LIN {X 0,Y 524.415,Z 426.256,A -85,B 0,C 180,E1 -4599.936,E2 -4599.936} C_VEL
LIN {X 0,Y 524.541,Z 418.004,A -85,B 0,C 180,E1 -4600.323,E2 -4600.323} C_VEL
LIN {X 0,Y 524.652,Z 409.12,A -85,B 0,C 180,E1 -4600.638,E2 -4600.638} C_VEL
LIN {X 0,Y 524.801,Z 400.246,A -85,B 0,C 180,E1 -4600.855,E2 -4600.855} C_VEL
LIN {X 0,Y 524.849,Z 331.396,A -85,B 0,C 180,E1 -4601.818,E2 -4601.818} C_VEL
LIN {X 0,Y 523.839,Z 323.933,A -85,B 0,C 180,E1 -4601.968,E2 -4601.968} C_VEL
LIN {X 0,Y 523.832,Z 321.449,A -85,B 0,C 180,E1 -4602.396,E2 -4602.396} C_VEL
LIN {X 0,Y 524.033,Z 307.521,A -85,B 0,C 180,E1 -4605.213,E2 -4605.213} C_VEL
LIN {X 0,Y 524.371,Z 292.162,A -85,B 0,C 180,E1 -4608.358,E2 -4608.358} C_VEL
LIN {X 0,Y 524.384,Z 283.062,A -85,B 0,C 180,E1 -4610.254,E2 -4610.254} C_VEL
LIN {X 0,Y 523.979,Z 280.14,A -85,B 0,C 180,E1 -4610.923,E2 -4610.923} C_VEL
LIN {X 0,Y 523.931,Z 280.033,A -85,B 0,C 180,E1 -4614.196,E2 -4614.196} C_VEL
LIN {X 0,Y 523.899,Z 280.036,A -85,B 0,C 180,E1 -4617.135,E2 -4617.135} C_VEL
LIN {X 0,Y 523.893,Z 280.04,A -85,B 0,C 180,E1 -4619.758,E2 -4619.758} C_VEL
LIN {X 0,Y 523.929,Z 280.029,A -85,B 0,C 180,E1 -4622.449,E2 -4622.449} C_VEL
LIN {X 0,Y 523.909,Z 280.038,A -85,B 0,C 180,E1 -4625.227,E2 -4625.227} C_VEL
LIN {X 0,Y 523.907,Z 280.033,A -85,B 0,C 180,E1 -4628.102,E2 -4628.102} C_VEL
LIN {X 0,Y 523.914,Z 280.04,A -85,B 0,C 180,E1 -4631.305,E2 -4631.305} C_VEL
LIN {X 0,Y 523.927,Z 280.032,A -85,B 0,C 180,E1 -4634.688,E2 -4634.688} C_VEL
LIN {X 0,Y 523.892,Z 280.035,A -85,B 0,C 180,E1 -4637.875,E2 -4637.875} C_VEL
LIN {X 0,Y 523.904,Z 280.041,A -85,B 0,C 180,E1 -4641.081,E2 -4641.081} C_VEL
LIN {X 0,Y 523.885,Z 280.035,A -85,B 0,C 180,E1 -4643.824,E2 -4643.824} C_VEL
LIN {X 0,Y 523.903,Z 280.038,A -85,B 0,C 180,E1 -4646.633,E2 -4646.633} C_VEL
LIN {X 0,Y 523.928,Z 280.031,A -85,B 0,C 180,E1 -4649.354,E2 -4649.354} C_VEL
LIN {X 0,Y 523.908,Z 280.035,A -85,B 0,C 180,E1 -4652.293,E2 -4652.293} C_VEL
LIN {X 0,Y 523.892,Z 280.035,A -85,B 0,C 180,E1 -4655.426,E2 -4655.426} C_VEL
LIN {X 0,Y 523.922,Z 280.032,A -85,B 0,C 180,E1 -4657.939,E2 -4657.939} C_VEL
LIN {X 0,Y 523.94,Z 280.036,A -85,B 0,C 180,E1 -4660.406,E2 -4660.406} C_VEL
LIN {X 0,Y 523.883,Z 280.039,A -85,B 0,C 180,E1 -4662.834,E2 -4662.834} C_VEL
LIN {X 0,Y 523.951,Z 280.027,A -85,B 0,C 180,E1 -4665.235,E2 -4665.235} C_VEL
LIN {X 0,Y 524.002,Z 280.028,A -85,B 0,C 180,E1 -4668.394,E2 -4668.394} C_VEL
LIN {X 0,Y 523.971,Z 280.025,A -85,B 0,C 180,E1 -4671.515,E2 -4671.515} C_VEL
LIN {X 0,Y 524.022,Z 280.021,A -85,B 0,C 180,E1 -4674.613,E2 -4674.613} C_VEL
LIN {X 0,Y 524.093,Z 280.013,A -85,B 0,C 180,E1 -4677.694,E2 -4677.694} C_VEL
LIN {X 0,Y 524.085,Z 280.019,A -85,B 0,C 180,E1 -4680,E2 -4680} C_VEL
LIN {X 0,Y 524.092,Z 280.013,A -85,B 0,C 180,E1 -4682.306,E2 -4682.306} C_VEL
LIN {X 0,Y 523.997,Z 280.026,A -85,B 0,C 180,E1 -4686.16,E2 -4686.16} C_VEL
LIN {X 0,Y 523.932,Z 280.031,A -85,B 0,C 180,E1 -4689.263,E2 -4689.263} C_VEL
LIN {X 0,Y 523.933,Z 280.03,A -85,B 0,C 180,E1 -4692.393,E2 -4692.393} C_VEL
LIN {X 0,Y 523.9,Z 280.041,A -85,B 0,C 180,E1 -4695.563,E2 -4695.563} C_VEL
LIN {X 0,Y 523.901,Z 280.036,A -85,B 0,C 180,E1 -4697.971,E2 -4697.971} C_VEL
LIN {X 0,Y 523.931,Z 280.029,A -85,B 0,C 180,E1 -4700.412,E2 -4700.412} C_VEL
LIN {X 0,Y 523.875,Z 280.038,A -85,B 0,C 180,E1 -4702.895,E2 -4702.895} C_VEL
LIN {X 0,Y 523.887,Z 280.043,A -85,B 0,C 180,E1 -4705.422,E2 -4705.422} C_VEL
LIN {X 0,Y 523.886,Z 280.036,A -85,B 0,C 180,E1 -4708.004,E2 -4708.004} C_VEL
LIN {X 0,Y 523.897,Z 280.037,A -85,B 0,C 180,E1 -4710.848,E2 -4710.848} C_VEL
LIN {X 0,Y 523.916,Z 280.033,A -85,B 0,C 180,E1 -4713.729,E2 -4713.729} C_VEL
LIN {X 0,Y 523.878,Z 280.037,A -85,B 0,C 180,E1 -4716.399,E2 -4716.399} C_VEL
LIN {X 0,Y 523.902,Z 280.042,A -85,B 0,C 180,E1 -4719.086,E2 -4719.086} C_VEL
LIN {X 0,Y 523.887,Z 280.035,A -85,B 0,C 180,E1 -4722.125,E2 -4722.125} C_VEL
LIN {X 0,Y 523.926,Z 280.033,A -85,B 0,C 180,E1 -4725.312,E2 -4725.312} C_VEL
LIN {X 0,Y 523.908,Z 280.04,A -85,B 0,C 180,E1 -4728.696,E2 -4728.696} C_VEL
LIN {X 0,Y 523.904,Z 280.033,A -85,B 0,C 180,E1 -4731.898,E2 -4731.898} C_VEL
LIN {X 0,Y 523.91,Z 280.037,A -85,B 0,C 180,E1 -4734.913,E2 -4734.913} C_VEL
LIN {X 0,Y 523.926,Z 280.03,A -85,B 0,C 180,E1 -4737.681,E2 -4737.681} C_VEL
LIN {X 0,Y 523.931,Z 280.036,A -85,B 0,C 180,E1 -4740.681,E2 -4740.681} C_VEL
LIN {X 0,Y 523.896,Z 280.034,A -85,B 0,C 180,E1 -4743.725,E2 -4743.725} C_VEL
LIN {X 0,Y 523.902,Z 280.034,A -85,B 0,C 180,E1 -4746.27,E2 -4746.27} C_VEL
LIN {X 0,Y 523.993,Z 280.189,A -85,B 0,C 180,E1 -4749.155,E2 -4749.155} C_VEL
LIN {X 0,Y 524.495,Z 286.09,A -85,B 0,C 180,E1 -4750.429,E2 -4750.429} C_VEL
LIN {X 0,Y 524.172,Z 299.754,A -85,B 0,C 180,E1 -4753.246,E2 -4753.246} C_VEL
LIN {X 0,Y 523.917,Z 313.418,A -85,B 0,C 180,E1 -4756.028,E2 -4756.028} C_VEL
LIN {X 0,Y 523.85,Z 323.715,A -85,B 0,C 180,E1 -4758.064,E2 -4758.064} C_VEL
LIN {X 0,Y 524.395,Z 328.212,A -85,B 0,C 180,E1 -4758.173,E2 -4758.173} C_VEL
LIN {X 0,Y 524.964,Z 334.33,A -85,B 0,C 180,E1 -4758.27,E2 -4758.27} C_VEL
LIN {X 0,Y 524.799,Z 399.153,A -85,B 0,C 180,E1 -4759.17,E2 -4759.17} C_VEL
LIN {X 0,Y 524.672,Z 408.418,A -85,B 0,C 180,E1 -4759.387,E2 -4759.387} C_VEL
LIN {X 0,Y 524.591,Z 416.888,A -85,B 0,C 180,E1 -4759.678,E2 -4759.678} C_VEL
LIN {X 0,Y 524.418,Z 425.391,A -85,B 0,C 180,E1 -4760.064,E2 -4760.064} C_VEL
LIN {X 0,Y 524.239,Z 433.724,A -85,B 0,C 180,E1 -4760.548,E2 -4760.548} C_VEL
LIN {X 0,Y 524.099,Z 441.761,A -85,B 0,C 180,E1 -4761.129,E2 -4761.129} C_VEL
LIN {X 0,Y 523.896,Z 450.433,A -85,B 0,C 180,E1 -4761.903,E2 -4761.903} C_VEL
LIN {X 0,Y 523.729,Z 458.939,A -85,B 0,C 180,E1 -4762.87,E2 -4762.87} C_VEL
LIN {X 0,Y 523.639,Z 465.61,A -85,B 0,C 180,E1 -4763.836,E2 -4763.836} C_VEL
LIN {X 0,Y 523.484,Z 469.989,A -85,B 0,C 180,E1 -4764.608,E2 -4764.608} C_VEL
LIN {X 0,Y 523.469,Z 475.15,A -85,B 0,C 180,E1 -4765.765,E2 -4765.765} C_VEL
LIN {X 0,Y 523.379,Z 478.938,A -85,B 0,C 180,E1 -4766.921,E2 -4766.921} C_VEL
LIN {X 0,Y 523.336,Z 480.68,A -85,B 0,C 180,E1 -4767.691,E2 -4767.691} C_VEL
LIN {X 0,Y 523.273,Z 481.928,A -85,B 0,C 180,E1 -4768.461,E2 -4768.461} C_VEL
LIN {X 0,Y 523.246,Z 482.706,A -85,B 0,C 180,E1 -4769.23,E2 -4769.23} C_VEL
LIN {X 0,Y 523.243,Z 483,A -85,B 0,C 180,E1 -4770,E2 -4770} C_VEL
LIN {X 0,Y 523.246,Z 482.705,A -85,B 0,C 180,E1 -4770.77,E2 -4770.77} C_VEL
LIN {X 0,Y 523.273,Z 481.927,A -85,B 0,C 180,E1 -4771.539,E2 -4771.539} C_VEL
LIN {X 0,Y 523.336,Z 480.679,A -85,B 0,C 180,E1 -4772.309,E2 -4772.309} C_VEL
LIN {X 0,Y 523.407,Z 477.786,A -85,B 0,C 180,E1 -4773.464,E2 -4773.464} C_VEL
LIN {X 0,Y 523.469,Z 475.149,A -85,B 0,C 180,E1 -4774.235,E2 -4774.235} C_VEL
LIN {X 0,Y 523.484,Z 469.986,A -85,B 0,C 180,E1 -4775.392,E2 -4775.392} C_VEL
LIN {X 0,Y 523.667,Z 463.738,A -85,B 0,C 180,E1 -4776.468,E2 -4776.468} C_VEL
LIN {X 0,Y 523.757,Z 455.74,A -85,B 0,C 180,E1 -4777.517,E2 -4777.517} C_VEL
LIN {X 0,Y 523.931,Z 448.398,A -85,B 0,C 180,E1 -4778.291,E2 -4778.291} C_VEL
LIN {X 0,Y 524.12,Z 440.535,A -85,B 0,C 180,E1 -4778.968,E2 -4778.968} C_VEL
LIN {X 0,Y 524.265,Z 432.224,A -85,B 0,C 180,E1 -4779.549,E2 -4779.549} C_VEL
LIN {X 0,Y 524.478,Z 421.614,A -85,B 0,C 180,E1 -4780.129,E2 -4780.129} C_VEL
LIN {X 0,Y 524.626,Z 410.084,A -85,B 0,C 180,E1 -4780.565,E2 -4780.565} C_VEL
LIN {X 0,Y 524.715,Z 400.451,A -85,B 0,C 180,E1 -4780.808,E2 -4780.808} C_VEL
LIN {X 0,Y 524.955,Z 348.572,A -85,B 0,C 180,E1 -4781.536,E2 -4781.536} C_VEL
LIN {X 0,Y 524.78,Z 330.794,A -85,B 0,C 180,E1 -4781.783,E2 -4781.783} C_VEL
LIN {X 0,Y 523.845,Z 323.822,A -85,B 0,C 180,E1 -4781.929,E2 -4781.929} C_VEL
LIN {X 0,Y 523.879,Z 317.322,A -85,B 0,C 180,E1 -4783.183,E2 -4783.183} C_VEL
LIN {X 0,Y 524.104,Z 303.658,A -85,B 0,C 180,E1 -4785.955,E2 -4785.955} C_VEL
LIN {X 0,Y 524.412,Z 289.994,A -85,B 0,C 180,E1 -4788.762,E2 -4788.762} C_VEL
LIN {X 0,Y 524.299,Z 282.187,A -85,B 0,C 180,E1 -4790.396,E2 -4790.396} C_VEL
LIN {X 0,Y 523.975,Z 280.145,A -85,B 0,C 180,E1 -4790.871,E2 -4790.871} C_VEL
LIN {X 0,Y 523.93,Z 280.033,A -85,B 0,C 180,E1 -4794.196,E2 -4794.196} C_VEL
LIN {X 0,Y 523.897,Z 280.037,A -85,B 0,C 180,E1 -4797.135,E2 -4797.135} C_VEL
LIN {X 0,Y 523.889,Z 280.039,A -85,B 0,C 180,E1 -4799.758,E2 -4799.758} C_VEL
LIN {X 0,Y 523.925,Z 280.03,A -85,B 0,C 180,E1 -4802.449,E2 -4802.449} C_VEL
LIN {X 0,Y 523.904,Z 280.04,A -85,B 0,C 180,E1 -4805.227,E2 -4805.227} C_VEL
LIN {X 0,Y 523.904,Z 280.033,A -85,B 0,C 180,E1 -4808.102,E2 -4808.102} C_VEL
LIN {X 0,Y 523.913,Z 280.039,A -85,B 0,C 180,E1 -4811.305,E2 -4811.305} C_VEL
LIN {X 0,Y 523.926,Z 280.033,A -85,B 0,C 180,E1 -4814.688,E2 -4814.688} C_VEL
LIN {X 0,Y 523.89,Z 280.035,A -85,B 0,C 180,E1 -4817.875,E2 -4817.875} C_VEL
LIN {X 0,Y 523.903,Z 280.04,A -85,B 0,C 180,E1 -4821.081,E2 -4821.081} C_VEL
LIN {X 0,Y 523.869,Z 280.037,A -85,B 0,C 180,E1 -4823.823,E2 -4823.823} C_VEL
LIN {X 0,Y 523.902,Z 280.039,A -85,B 0,C 180,E1 -4826.633,E2 -4826.633} C_VEL
LIN {X 0,Y 523.927,Z 280.031,A -85,B 0,C 180,E1 -4829.354,E2 -4829.354} C_VEL
LIN {X 0,Y 523.907,Z 280.036,A -85,B 0,C 180,E1 -4832.294,E2 -4832.294} C_VEL
LIN {X 0,Y 523.891,Z 280.035,A -85,B 0,C 180,E1 -4835.426,E2 -4835.426} C_VEL
LIN {X 0,Y 523.921,Z 280.032,A -85,B 0,C 180,E1 -4837.939,E2 -4837.939} C_VEL
LIN {X 0,Y 523.94,Z 280.036,A -85,B 0,C 180,E1 -4840.407,E2 -4840.407} C_VEL
LIN {X 0,Y 523.882,Z 280.039,A -85,B 0,C 180,E1 -4842.834,E2 -4842.834} C_VEL
LIN {X 0,Y 523.951,Z 280.027,A -85,B 0,C 180,E1 -4845.235,E2 -4845.235} C_VEL
LIN {X 0,Y 524.002,Z 280.028,A -85,B 0,C 180,E1 -4848.394,E2 -4848.394} C_VEL
LIN {X 0,Y 523.941,Z 280.029,A -85,B 0,C 180,E1 -4851.515,E2 -4851.515} C_VEL
LIN {X 0,Y 524.022,Z 280.021,A -85,B 0,C 180,E1 -4854.613,E2 -4854.613} C_VEL
LIN {X 0,Y 524.093,Z 280.013,A -85,B 0,C 180,E1 -4857.694,E2 -4857.694} C_VEL
LIN {X 0,Y 524.085,Z 280.019,A -85,B 0,C 180,E1 -4860,E2 -4860} C_VEL
LIN {X 0,Y 524.092,Z 280.013,A -85,B 0,C 180,E1 -4862.306,E2 -4862.306} C_VEL
LIN {X 0,Y 523.997,Z 280.026,A -85,B 0,C 180,E1 -4866.16,E2 -4866.16} C_VEL
LIN {X 0,Y 523.932,Z 280.031,A -85,B 0,C 180,E1 -4869.263,E2 -4869.263} C_VEL
LIN {X 0,Y 523.933,Z 280.03,A -85,B 0,C 180,E1 -4872.393,E2 -4872.393} C_VEL
LIN {X 0,Y 523.9,Z 280.041,A -85,B 0,C 180,E1 -4875.563,E2 -4875.563} C_VEL
LIN {X 0,Y 523.913,Z 280.032,A -85,B 0,C 180,E1 -4878.781,E2 -4878.781} C_VEL
LIN {X 0,Y 523.911,Z 280.037,A -85,B 0,C 180,E1 -4881.235,E2 -4881.235} C_VEL
LIN {X 0,Y 523.891,Z 280.034,A -85,B 0,C 180,E1 -4884.574,E2 -4884.574} C_VEL
LIN {X 0,Y 523.901,Z 280.037,A -85,B 0,C 180,E1 -4887.705,E2 -4887.705} C_VEL
LIN {X 0,Y 523.899,Z 280.035,A -85,B 0,C 180,E1 -4890.648,E2 -4890.648} C_VEL
LIN {X 0,Y 523.903,Z 280.039,A -85,B 0,C 180,E1 -4893.367,E2 -4893.367} C_VEL
LIN {X 0,Y 523.878,Z 280.036,A -85,B 0,C 180,E1 -4896.399,E2 -4896.399} C_VEL
LIN {X 0,Y 523.902,Z 280.042,A -85,B 0,C 180,E1 -4899.087,E2 -4899.087} C_VEL
LIN {X 0,Y 523.888,Z 280.035,A -85,B 0,C 180,E1 -4902.125,E2 -4902.125} C_VEL
LIN {X 0,Y 523.927,Z 280.033,A -85,B 0,C 180,E1 -4905.312,E2 -4905.312} C_VEL
LIN {X 0,Y 523.872,Z 280.044,A -85,B 0,C 180,E1 -4906.871,E2 -4906.871} C_VEL
LIN {X 0,Y 523.184,Z 280.125,A -85,B 0,C 180,E1 -4907.512,E2 -4907.512} C_VEL
LIN {X 0,Y 520.321,Z 280.484,A -85,B 0,C 180,E1 -4908.554,E2 -4908.554} C_VEL
LIN {X 0,Y 517.928,Z 280.779,A -85,B 0,C 180,E1 -4909.392,E2 -4909.392} C_VEL
LIN {X 0,Y 516.922,Z 280.903,A -85,B 0,C 180,E1 -4910.04,E2 -4910.04} C_VEL
LIN {X 0,Y 516.851,Z 280.913,A -85,B 0,C 180,E1 -4910.259,E2 -4910.259} C_VEL
LIN {X 0,Y 516.845,Z 280.914,A -85,B 0,C 180,E1 -4913.252,E2 -4913.252} C_VEL
LIN {X 0,Y 516.875,Z 280.91,A -85,B 0,C 180,E1 -4916.119,E2 -4916.119} C_VEL
LIN {X 0,Y 516.875,Z 280.912,A -85,B 0,C 180,E1 -4918.939,E2 -4918.939} C_VEL
LIN {X 0,Y 516.858,Z 280.914,A -85,B 0,C 180,E1 -4922.109,E2 -4922.109} C_VEL
LIN {X 0,Y 516.843,Z 280.915,A -85,B 0,C 180,E1 -4925.069,E2 -4925.069} C_VEL
LIN {X 0,Y 516.869,Z 280.898,A -85,B 0,C 180,E1 -4927.622,E2 -4927.622} C_VEL
LIN {X 0,Y 516.925,Z 281.074,A -85,B 0,C 180,E1 -4929.091,E2 -4929.091} C_VEL
LIN {X 0,Y 517.472,Z 285.88,A -85,B 0,C 180,E1 -4930.152,E2 -4930.152} C_VEL
LIN {X 0,Y 517.255,Z 297.588,A -85,B 0,C 180,E1 -4932.608,E2 -4932.608} C_VEL
LIN {X 0,Y 516.908,Z 313.2,A -85,B 0,C 180,E1 -4935.834,E2 -4935.834} C_VEL
LIN {X 0,Y 516.779,Z 323.603,A -85,B 0,C 180,E1 -4937.928,E2 -4937.928} C_VEL
LIN {X 0,Y 516.978,Z 325.468,A -85,B 0,C 180,E1 -4938.008,E2 -4938.008} C_VEL
LIN {X 0,Y 518.064,Z 333.866,A -85,B 0,C 180,E1 -4938.15,E2 -4938.15} C_VEL
LIN {X 0,Y 517.841,Z 399.389,A -85,B 0,C 180,E1 -4939.072,E2 -4939.072} C_VEL
LIN {X 0,Y 517.699,Z 408.571,A -85,B 0,C 180,E1 -4939.292,E2 -4939.292} C_VEL
LIN {X 0,Y 517.566,Z 418.209,A -85,B 0,C 180,E1 -4939.635,E2 -4939.635} C_VEL
LIN {X 0,Y 517.426,Z 428.284,A -85,B 0,C 180,E1 -4940.126,E2 -4940.126} C_VEL
LIN {X 0,Y 517.146,Z 438.743,A -85,B 0,C 180,E1 -4940.812,E2 -4940.812} C_VEL
LIN {X 0,Y 516.908,Z 446.911,A -85,B 0,C 180,E1 -4941.497,E2 -4941.497} C_VEL
LIN {X 0,Y 516.744,Z 453.65,A -85,B 0,C 180,E1 -4942.183,E2 -4942.183} C_VEL
LIN {X 0,Y 516.66,Z 460.03,A -85,B 0,C 180,E1 -4942.968,E2 -4942.968} C_VEL
LIN {X 0,Y 516.585,Z 465.335,A -85,B 0,C 180,E1 -4943.752,E2 -4943.752} C_VEL
LIN {X 0,Y 516.434,Z 469.766,A -85,B 0,C 180,E1 -4944.534,E2 -4944.534} C_VEL
LIN {X 0,Y 516.322,Z 473.458,A -85,B 0,C 180,E1 -4945.316,E2 -4945.316} C_VEL
LIN {X 0,Y 516.386,Z 476.469,A -85,B 0,C 180,E1 -4946.098,E2 -4946.098} C_VEL
LIN {X 0,Y 516.295,Z 478.804,A -85,B 0,C 180,E1 -4946.879,E2 -4946.879} C_VEL
LIN {X 0,Y 516.263,Z 480.586,A -85,B 0,C 180,E1 -4947.659,E2 -4947.659} C_VEL
LIN {X 0,Y 516.19,Z 481.872,A -85,B 0,C 180,E1 -4948.44,E2 -4948.44} C_VEL
LIN {X 0,Y 516.157,Z 482.687,A -85,B 0,C 180,E1 -4949.22,E2 -4949.22} C_VEL
LIN {X 0,Y 516.152,Z 482.997,A -85,B 0,C 180,E1 -4950,E2 -4950} C_VEL
LIN {X 0,Y 516.157,Z 482.724,A -85,B 0,C 180,E1 -4950.78,E2 -4950.78} C_VEL
LIN {X 0,Y 516.191,Z 481.984,A -85,B 0,C 180,E1 -4951.56,E2 -4951.56} C_VEL
LIN {X 0,Y 516.264,Z 480.773,A -85,B 0,C 180,E1 -4952.341,E2 -4952.341} C_VEL
LIN {X 0,Y 516.324,Z 477.919,A -85,B 0,C 180,E1 -4953.512,E2 -4953.512} C_VEL
LIN {X 0,Y 516.39,Z 475.324,A -85,B 0,C 180,E1 -4954.293,E2 -4954.293} C_VEL
LIN {X 0,Y 516.431,Z 470.209,A -85,B 0,C 180,E1 -4955.466,E2 -4955.466} C_VEL
LIN {X 0,Y 516.572,Z 464.572,A -85,B 0,C 180,E1 -4956.467,E2 -4956.467} C_VEL
LIN {X 0,Y 516.683,Z 457.804,A -85,B 0,C 180,E1 -4957.424,E2 -4957.424} C_VEL
LIN {X 0,Y 516.886,Z 448.858,A -85,B 0,C 180,E1 -4958.405,E2 -4958.405} C_VEL
LIN {X 0,Y 517.093,Z 441.093,A -85,B 0,C 180,E1 -4959.091,E2 -4959.091} C_VEL
LIN {X 0,Y 517.262,Z 432.907,A -85,B 0,C 180,E1 -4959.679,E2 -4959.679} C_VEL
LIN {X 0,Y 517.467,Z 424.371,A -85,B 0,C 180,E1 -4960.169,E2 -4960.169} C_VEL
LIN {X 0,Y 517.648,Z 414.36,A -85,B 0,C 180,E1 -4960.61,E2 -4960.61} C_VEL
LIN {X 0,Y 517.767,Z 402.807,A -85,B 0,C 180,E1 -4960.954,E2 -4960.954} C_VEL
LIN {X 0,Y 517.927,Z 384.017,A -85,B 0,C 180,E1 -4961.248,E2 -4961.248} C_VEL
LIN {X 0,Y 517.868,Z 332.03,A -85,B 0,C 180,E1 -4961.97,E2 -4961.97} C_VEL
LIN {X 0,Y 516.82,Z 324.148,A -85,B 0,C 180,E1 -4962.123,E2 -4962.123} C_VEL
LIN {X 0,Y 516.777,Z 323.53,A -85,B 0,C 180,E1 -4962.169,E2 -4962.169} C_VEL
LIN {X 0,Y 517.026,Z 307.635,A -85,B 0,C 180,E1 -4965.4,E2 -4965.4} C_VEL
LIN {X 0,Y 517.394,Z 292.158,A -85,B 0,C 180,E1 -4968.615,E2 -4968.615} C_VEL
LIN {X 0,Y 517.352,Z 283.764,A -85,B 0,C 180,E1 -4970.391,E2 -4970.391} C_VEL
LIN {X 0,Y 516.948,Z 281.03,A -85,B 0,C 180,E1 -4971.012,E2 -4971.012} C_VEL
LIN {X 0,Y 516.871,Z 280.912,A -85,B 0,C 180,E1 -4974.354,E2 -4974.354} C_VEL
LIN {X 0,Y 516.84,Z 280.913,A -85,B 0,C 180,E1 -4976.662,E2 -4976.662} C_VEL
LIN {X 0,Y 516.883,Z 280.916,A -85,B 0,C 180,E1 -4979.518,E2 -4979.518} C_VEL
LIN {X 0,Y 516.89,Z 280.906,A -85,B 0,C 180,E1 -4982.542,E2 -4982.542} C_VEL
LIN {X 0,Y 516.856,Z 280.919,A -85,B 0,C 180,E1 -4985.328,E2 -4985.328} C_VEL
LIN {X 0,Y 516.872,Z 280.91,A -85,B 0,C 180,E1 -4987.942,E2 -4987.942} C_VEL
LIN {X 0,Y 516.847,Z 280.914,A -85,B 0,C 180,E1 -4990.744,E2 -4990.744} C_VEL
LIN {X 0,Y 516.874,Z 280.909,A -85,B 0,C 180,E1 -4993.903,E2 -4993.903} C_VEL
LIN {X 0,Y 516.873,Z 280.908,A -85,B 0,C 180,E1 -4996.107,E2 -4996.107} C_VEL
LIN {X 0,Y 516.845,Z 280.918,A -85,B 0,C 180,E1 -4999.255,E2 -4999.255} C_VEL
LIN {X 0,Y 516.852,Z 280.912,A -85,B 0,C 180,E1 -5002.273,E2 -5002.273} C_VEL
LIN {X 0,Y 516.864,Z 280.915,A -85,B 0,C 180,E1 -5005.174,E2 -5005.174} C_VEL
LIN {X 0,Y 516.858,Z 280.911,A -85,B 0,C 180,E1 -5007.974,E2 -5007.974} C_VEL
LIN {X 0,Y 516.893,Z 280.914,A -85,B 0,C 180,E1 -5010.694,E2 -5010.694} C_VEL
LIN {X 0,Y 516.872,Z 280.909,A -85,B 0,C 180,E1 -5013.817,E2 -5013.817} C_VEL
LIN {X 0,Y 516.841,Z 280.919,A -85,B 0,C 180,E1 -5016.775,E2 -5016.775} C_VEL
LIN {X 0,Y 516.896,Z 280.906,A -85,B 0,C 180,E1 -5019.741,E2 -5019.741} C_VEL
LIN {X 0,Y 516.853,Z 280.918,A -85,B 0,C 180,E1 -5022.593,E2 -5022.593} C_VEL
LIN {X 0,Y 516.92,Z 280.904,A -85,B 0,C 180,E1 -5025.029,E2 -5025.029} C_VEL
LIN {X 0,Y 516.956,Z 280.906,A -85,B 0,C 180,E1 -5028.233,E2 -5028.233} C_VEL
LIN {X 0,Y 516.939,Z 280.901,A -85,B 0,C 180,E1 -5031.399,E2 -5031.399} C_VEL
LIN {X 0,Y 516.973,Z 280.9,A -85,B 0,C 180,E1 -5034.539,E2 -5034.539} C_VEL
LIN {X 0,Y 517.062,Z 280.888,A -85,B 0,C 180,E1 -5037.663,E2 -5037.663} C_VEL
LIN {X 0,Y 517.053,Z 280.895,A -85,B 0,C 180,E1 -5040,E2 -5040} C_VEL
LIN {X 0,Y 517.061,Z 280.889,A -85,B 0,C 180,E1 -5042.337,E2 -5042.337} C_VEL
LIN {X 0,Y 516.962,Z 280.901,A -85,B 0,C 180,E1 -5046.244,E2 -5046.244} C_VEL
LIN {X 0,Y 516.895,Z 280.909,A -85,B 0,C 180,E1 -5049.39,E2 -5049.39} C_VEL
LIN {X 0,Y 516.885,Z 280.907,A -85,B 0,C 180,E1 -5052.565,E2 -5052.565} C_VEL
LIN {X 0,Y 516.925,Z 280.904,A -85,B 0,C 180,E1 -5055.143,E2 -5055.143} C_VEL
LIN {X 0,Y 516.862,Z 280.911,A -85,B 0,C 180,E1 -5058.224,E2 -5058.224} C_VEL
LIN {X 0,Y 516.879,Z 280.908,A -85,B 0,C 180,E1 -5060.703,E2 -5060.703} C_VEL
LIN {X 0,Y 516.83,Z 280.92,A -85,B 0,C 180,E1 -5063.225,E2 -5063.225} C_VEL
LIN {X 0,Y 516.868,Z 280.909,A -85,B 0,C 180,E1 -5066.182,E2 -5066.182} C_VEL
LIN {X 0,Y 516.874,Z 280.914,A -85,B 0,C 180,E1 -5069.519,E2 -5069.519} C_VEL
LIN {X 0,Y 516.882,Z 280.908,A -85,B 0,C 180,E1 -5072.543,E2 -5072.543} C_VEL
LIN {X 0,Y 516.845,Z 280.918,A -85,B 0,C 180,E1 -5075.328,E2 -5075.328} C_VEL
LIN {X 0,Y 516.868,Z 280.909,A -85,B 0,C 180,E1 -5077.943,E2 -5077.943} C_VEL
LIN {X 0,Y 516.843,Z 280.917,A -85,B 0,C 180,E1 -5080.745,E2 -5080.745} C_VEL
LIN {X 0,Y 516.873,Z 280.909,A -85,B 0,C 180,E1 -5083.904,E2 -5083.904} C_VEL
LIN {X 0,Y 516.873,Z 280.909,A -85,B 0,C 180,E1 -5086.108,E2 -5086.108} C_VEL
LIN {X 0,Y 516.843,Z 280.915,A -85,B 0,C 180,E1 -5089.256,E2 -5089.256} C_VEL
LIN {X 0,Y 516.853,Z 280.914,A -85,B 0,C 180,E1 -5092.274,E2 -5092.274} C_VEL
LIN {X 0,Y 516.866,Z 280.911,A -85,B 0,C 180,E1 -5095.175,E2 -5095.175} C_VEL
LIN {X 0,Y 516.862,Z 280.911,A -85,B 0,C 180,E1 -5097.975,E2 -5097.975} C_VEL
LIN {X 0,Y 516.899,Z 280.911,A -85,B 0,C 180,E1 -5100.695,E2 -5100.695} C_VEL
LIN {X 0,Y 516.876,Z 280.91,A -85,B 0,C 180,E1 -5103.819,E2 -5103.819} C_VEL
LIN {X 0,Y 516.849,Z 280.903,A -85,B 0,C 180,E1 -5106.776,E2 -5106.776} C_VEL
LIN {X 0,Y 516.945,Z 281.051,A -85,B 0,C 180,E1 -5109.04,E2 -5109.04} C_VEL
LIN {X 0,Y 517.498,Z 286.09,A -85,B 0,C 180,E1 -5110.153,E2 -5110.153} C_VEL
LIN {X 0,Y 517.186,Z 299.754,A -85,B 0,C 180,E1 -5113.013,E2 -5113.013} C_VEL
LIN {X 0,Y 516.907,Z 313.418,A -85,B 0,C 180,E1 -5115.834,E2 -5115.834} C_VEL
LIN {X 0,Y 516.816,Z 323.726,A -85,B 0,C 180,E1 -5117.899,E2 -5117.899} C_VEL
LIN {X 0,Y 517.405,Z 328.439,A -85,B 0,C 180,E1 -5118.014,E2 -5118.014} C_VEL
LIN {X 0,Y 518.041,Z 335.147,A -85,B 0,C 180,E1 -5118.122,E2 -5118.122} C_VEL
LIN {X 0,Y 517.839,Z 399.187,A -85,B 0,C 180,E1 -5119.023,E2 -5119.023} C_VEL
LIN {X 0,Y 517.708,Z 408.418,A -85,B 0,C 180,E1 -5119.242,E2 -5119.242} C_VEL
LIN {X 0,Y 517.593,Z 416.888,A -85,B 0,C 180,E1 -5119.537,E2 -5119.537} C_VEL
LIN {X 0,Y 517.411,Z 425.391,A -85,B 0,C 180,E1 -5119.928,E2 -5119.928} C_VEL
LIN {X 0,Y 517.243,Z 433.724,A -85,B 0,C 180,E1 -5120.419,E2 -5120.419} C_VEL
LIN {X 0,Y 517.084,Z 441.761,A -85,B 0,C 180,E1 -5121.008,E2 -5121.008} C_VEL
LIN {X 0,Y 516.846,Z 450.433,A -85,B 0,C 180,E1 -5121.792,E2 -5121.792} C_VEL
LIN {X 0,Y 516.659,Z 458.939,A -85,B 0,C 180,E1 -5122.772,E2 -5122.772} C_VEL
LIN {X 0,Y 516.575,Z 465.61,A -85,B 0,C 180,E1 -5123.752,E2 -5123.752} C_VEL
LIN {X 0,Y 516.431,Z 469.989,A -85,B 0,C 180,E1 -5124.534,E2 -5124.534} C_VEL
LIN {X 0,Y 516.392,Z 475.15,A -85,B 0,C 180,E1 -5125.707,E2 -5125.707} C_VEL
LIN {X 0,Y 516.324,Z 477.787,A -85,B 0,C 180,E1 -5126.488,E2 -5126.488} C_VEL
LIN {X 0,Y 516.262,Z 480.68,A -85,B 0,C 180,E1 -5127.659,E2 -5127.659} C_VEL
LIN {X 0,Y 516.19,Z 481.928,A -85,B 0,C 180,E1 -5128.44,E2 -5128.44} C_VEL
LIN {X 0,Y 516.156,Z 482.706,A -85,B 0,C 180,E1 -5129.22,E2 -5129.22} C_VEL
LIN {X 0,Y 516.151,Z 483,A -85,B 0,C 180,E1 -5130,E2 -5130} C_VEL
LIN {X 0,Y 516.156,Z 482.705,A -85,B 0,C 180,E1 -5130.78,E2 -5130.78} C_VEL
LIN {X 0,Y 516.19,Z 481.927,A -85,B 0,C 180,E1 -5131.56,E2 -5131.56} C_VEL
LIN {X 0,Y 516.262,Z 480.679,A -85,B 0,C 180,E1 -5132.341,E2 -5132.341} C_VEL
LIN {X 0,Y 516.324,Z 477.786,A -85,B 0,C 180,E1 -5133.512,E2 -5133.512} C_VEL
LIN {X 0,Y 516.392,Z 475.149,A -85,B 0,C 180,E1 -5134.293,E2 -5134.293} C_VEL
LIN {X 0,Y 516.431,Z 469.986,A -85,B 0,C 180,E1 -5135.466,E2 -5135.466} C_VEL
LIN {X 0,Y 516.58,Z 464.233,A -85,B 0,C 180,E1 -5136.478,E2 -5136.478} C_VEL
LIN {X 0,Y 516.685,Z 457.436,A -85,B 0,C 180,E1 -5137.424,E2 -5137.424} C_VEL
LIN {X 0,Y 516.862,Z 449.419,A -85,B 0,C 180,E1 -5138.307,E2 -5138.307} C_VEL
LIN {X 0,Y 517.084,Z 441.765,A -85,B 0,C 180,E1 -5138.992,E2 -5138.992} C_VEL
LIN {X 0,Y 517.243,Z 433.725,A -85,B 0,C 180,E1 -5139.581,E2 -5139.581} C_VEL
LIN {X 0,Y 517.411,Z 425.393,A -85,B 0,C 180,E1 -5140.072,E2 -5140.072} C_VEL
LIN {X 0,Y 517.593,Z 416.891,A -85,B 0,C 180,E1 -5140.463,E2 -5140.463} C_VEL
LIN {X 0,Y 517.692,Z 407.589,A -85,B 0,C 180,E1 -5140.783,E2 -5140.783} C_VEL
LIN {X 0,Y 517.88,Z 396.668,A -85,B 0,C 180,E1 -5141.024,E2 -5141.024} C_VEL
LIN {X 0,Y 517.877,Z 331.791,A -85,B 0,C 180,E1 -5141.928,E2 -5141.928} C_VEL
LIN {X 0,Y 516.806,Z 323.959,A -85,B 0,C 180,E1 -5142.083,E2 -5142.083} C_VEL
LIN {X 0,Y 516.794,Z 321.226,A -85,B 0,C 180,E1 -5142.567,E2 -5142.567} C_VEL
LIN {X 0,Y 517.056,Z 305.61,A -85,B 0,C 180,E1 -5145.774,E2 -5145.774} C_VEL
LIN {X 0,Y 517.4,Z 291.946,A -85,B 0,C 180,E1 -5148.615,E2 -5148.615} C_VEL
LIN {X 0,Y 517.329,Z 283.59,A -85,B 0,C 180,E1 -5150.385,E2 -5150.385} C_VEL
LIN {X 0,Y 516.918,Z 281.001,A -85,B 0,C 180,E1 -5151.013,E2 -5151.013} C_VEL
LIN {X 0,Y 516.869,Z 280.912,A -85,B 0,C 180,E1 -5154.354,E2 -5154.354} C_VEL
LIN {X 0,Y 516.839,Z 280.913,A -85,B 0,C 180,E1 -5156.662,E2 -5156.662} C_VEL
LIN {X 0,Y 516.881,Z 280.916,A -85,B 0,C 180,E1 -5159.518,E2 -5159.518} C_VEL
LIN {X 0,Y 516.887,Z 280.907,A -85,B 0,C 180,E1 -5162.542,E2 -5162.542} C_VEL
LIN {X 0,Y 516.849,Z 280.92,A -85,B 0,C 180,E1 -5165.327,E2 -5165.327} C_VEL
LIN {X 0,Y 516.87,Z 280.91,A -85,B 0,C 180,E1 -5167.942,E2 -5167.942} C_VEL
LIN {X 0,Y 516.846,Z 280.914,A -85,B 0,C 180,E1 -5170.744,E2 -5170.744} C_VEL
LIN {X 0,Y 516.873,Z 280.909,A -85,B 0,C 180,E1 -5173.903,E2 -5173.903} C_VEL
LIN {X 0,Y 516.872,Z 280.909,A -85,B 0,C 180,E1 -5176.107,E2 -5176.107} C_VEL
LIN {X 0,Y 516.844,Z 280.917,A -85,B 0,C 180,E1 -5179.255,E2 -5179.255} C_VEL
LIN {X 0,Y 516.851,Z 280.912,A -85,B 0,C 180,E1 -5182.273,E2 -5182.273} C_VEL
LIN {X 0,Y 516.862,Z 280.914,A -85,B 0,C 180,E1 -5185.174,E2 -5185.174} C_VEL
LIN {X 0,Y 516.857,Z 280.911,A -85,B 0,C 180,E1 -5187.974,E2 -5187.974} C_VEL
LIN {X 0,Y 516.892,Z 280.915,A -85,B 0,C 180,E1 -5190.694,E2 -5190.694} C_VEL
LIN {X 0,Y 516.871,Z 280.909,A -85,B 0,C 180,E1 -5193.818,E2 -5193.818} C_VEL
LIN {X 0,Y 516.841,Z 280.919,A -85,B 0,C 180,E1 -5196.775,E2 -5196.775} C_VEL
LIN {X 0,Y 516.896,Z 280.906,A -85,B 0,C 180,E1 -5199.741,E2 -5199.741} C_VEL
LIN {X 0,Y 516.853,Z 280.918,A -85,B 0,C 180,E1 -5202.594,E2 -5202.594} C_VEL
LIN {X 0,Y 516.92,Z 280.904,A -85,B 0,C 180,E1 -5205.03,E2 -5205.03} C_VEL
LIN {X 0,Y 516.955,Z 280.906,A -85,B 0,C 180,E1 -5208.234,E2 -5208.234} C_VEL
LIN {X 0,Y 516.917,Z 280.903,A -85,B 0,C 180,E1 -5211.399,E2 -5211.399} C_VEL
LIN {X 0,Y 516.973,Z 280.9,A -85,B 0,C 180,E1 -5214.539,E2 -5214.539} C_VEL
LIN {X 0,Y 517.062,Z 280.888,A -85,B 0,C 180,E1 -5217.663,E2 -5217.663} C_VEL
LIN {X 0,Y 517.053,Z 280.895,A -85,B 0,C 180,E1 -5220,E2 -5220} C_VEL
LIN {X 0,Y 517.061,Z 280.889,A -85,B 0,C 180,E1 -5222.337,E2 -5222.337} C_VEL
LIN {X 0,Y 516.963,Z 280.901,A -85,B 0,C 180,E1 -5226.244,E2 -5226.244} C_VEL
LIN {X 0,Y 516.894,Z 280.909,A -85,B 0,C 180,E1 -5229.39,E2 -5229.39} C_VEL
LIN {X 0,Y 516.885,Z 280.907,A -85,B 0,C 180,E1 -5232.565,E2 -5232.565} C_VEL
LIN {X 0,Y 516.924,Z 280.904,A -85,B 0,C 180,E1 -5235.142,E2 -5235.142} C_VEL
LIN {X 0,Y 516.862,Z 280.911,A -85,B 0,C 180,E1 -5238.225,E2 -5238.225} C_VEL
LIN {X 0,Y 516.879,Z 280.908,A -85,B 0,C 180,E1 -5240.703,E2 -5240.703} C_VEL
LIN {X 0,Y 516.83,Z 280.919,A -85,B 0,C 180,E1 -5243.226,E2 -5243.226} C_VEL
LIN {X 0,Y 516.869,Z 280.909,A -85,B 0,C 180,E1 -5246.182,E2 -5246.182} C_VEL
LIN {X 0,Y 516.887,Z 280.916,A -85,B 0,C 180,E1 -5249.307,E2 -5249.307} C_VEL
LIN {X 0,Y 516.883,Z 280.908,A -85,B 0,C 180,E1 -5252.543,E2 -5252.543} C_VEL
LIN {X 0,Y 516.845,Z 280.918,A -85,B 0,C 180,E1 -5255.328,E2 -5255.328} C_VEL
LIN {X 0,Y 516.868,Z 280.909,A -85,B 0,C 180,E1 -5257.943,E2 -5257.943} C_VEL
LIN {X 0,Y 516.843,Z 280.917,A -85,B 0,C 180,E1 -5260.746,E2 -5260.746} C_VEL
LIN {X 0,Y 516.874,Z 280.908,A -85,B 0,C 180,E1 -5263.904,E2 -5263.904} C_VEL
LIN {X 0,Y 516.828,Z 280.915,A -85,B 0,C 180,E1 -5266.87,E2 -5266.87} C_VEL
LIN {X 0,Y 516.853,Z 280.911,A -85,B 0,C 180,E1 -5269.594,E2 -5269.594} C_VEL
LIN {X 0,Y 516.851,Z 280.913,A -85,B 0,C 180,E1 -5270.259,E2 -5270.259} C_VEL
LIN {X 0,Y 516.215,Z 280.998,A -85,B 0,C 180,E1 -5270.91,E2 -5270.91} C_VEL
LIN {X 0,Y 513.369,Z 281.351,A -85,B 0,C 180,E1 -5271.965,E2 -5271.965} C_VEL
LIN {X 0,Y 510.939,Z 281.655,A -85,B 0,C 180,E1 -5272.815,E2 -5272.815} C_VEL
LIN {X 0,Y 509.886,Z 281.78,A -85,B 0,C 180,E1 -5273.472,E2 -5273.472} C_VEL
LIN {X 0,Y 509.796,Z 281.79,A -85,B 0,C 180,E1 -5273.694,E2 -5273.694} C_VEL
LIN {X 0,Y 509.835,Z 281.793,A -85,B 0,C 180,E1 -5276.538,E2 -5276.538} C_VEL
LIN {X 0,Y 509.814,Z 281.788,A -85,B 0,C 180,E1 -5279.333,E2 -5279.333} C_VEL
LIN {X 0,Y 509.825,Z 281.789,A -85,B 0,C 180,E1 -5282.051,E2 -5282.051} C_VEL
LIN {X 0,Y 509.799,Z 281.797,A -85,B 0,C 180,E1 -5284.701,E2 -5284.701} C_VEL
LIN {X 0,Y 509.822,Z 281.775,A -85,B 0,C 180,E1 -5287.46,E2 -5287.46} C_VEL
LIN {X 0,Y 509.882,Z 282.02,A -85,B 0,C 180,E1 -5289,E2 -5289} C_VEL
LIN {X 0,Y 510.48,Z 287.834,A -85,B 0,C 180,E1 -5290.288,E2 -5290.288} C_VEL
LIN {X 0,Y 510.146,Z 301.494,A -85,B 0,C 180,E1 -5293.184,E2 -5293.184} C_VEL
LIN {X 0,Y 509.826,Z 315.155,A -85,B 0,C 180,E1 -5296.041,E2 -5296.041} C_VEL
LIN {X 0,Y 509.741,Z 323.68,A -85,B 0,C 180,E1 -5297.766,E2 -5297.766} C_VEL
LIN {X 0,Y 510.25,Z 327.434,A -85,B 0,C 180,E1 -5297.874,E2 -5297.874} C_VEL
LIN {X 0,Y 511.113,Z 335.298,A -85,B 0,C 180,E1 -5298.006,E2 -5298.006} C_VEL
LIN {X 0,Y 510.898,Z 399.422,A -85,B 0,C 180,E1 -5298.922,E2 -5298.922} C_VEL
LIN {X 0,Y 510.735,Z 408.592,A -85,B 0,C 180,E1 -5299.144,E2 -5299.144} C_VEL
LIN {X 0,Y 510.594,Z 418.225,A -85,B 0,C 180,E1 -5299.492,E2 -5299.492} C_VEL
LIN {X 0,Y 510.443,Z 426.424,A -85,B 0,C 180,E1 -5299.89,E2 -5299.89} C_VEL
LIN {X 0,Y 510.207,Z 436.05,A -85,B 0,C 180,E1 -5300.486,E2 -5300.486} C_VEL
LIN {X 0,Y 509.916,Z 445.896,A -85,B 0,C 180,E1 -5301.28,E2 -5301.28} C_VEL
LIN {X 0,Y 509.711,Z 453.655,A -85,B 0,C 180,E1 -5302.075,E2 -5302.075} C_VEL
LIN {X 0,Y 509.609,Z 460.035,A -85,B 0,C 180,E1 -5302.87,E2 -5302.87} C_VEL
LIN {X 0,Y 509.503,Z 466.512,A -85,B 0,C 180,E1 -5303.863,E2 -5303.863} C_VEL
LIN {X 0,Y 509.282,Z 471.682,A -85,B 0,C 180,E1 -5304.854,E2 -5304.854} C_VEL
LIN {X 0,Y 509.301,Z 476.471,A -85,B 0,C 180,E1 -5306.044,E2 -5306.044} C_VEL
LIN {X 0,Y 509.213,Z 478.806,A -85,B 0,C 180,E1 -5306.835,E2 -5306.835} C_VEL
LIN {X 0,Y 509.192,Z 480.587,A -85,B 0,C 180,E1 -5307.627,E2 -5307.627} C_VEL
LIN {X 0,Y 509.111,Z 481.873,A -85,B 0,C 180,E1 -5308.418,E2 -5308.418} C_VEL
LIN {X 0,Y 509.07,Z 482.687,A -85,B 0,C 180,E1 -5309.209,E2 -5309.209} C_VEL
LIN {X 0,Y 509.063,Z 482.997,A -85,B 0,C 180,E1 -5310,E2 -5310} C_VEL
LIN {X 0,Y 509.071,Z 482.724,A -85,B 0,C 180,E1 -5310.791,E2 -5310.791} C_VEL
LIN {X 0,Y 509.112,Z 481.983,A -85,B 0,C 180,E1 -5311.582,E2 -5311.582} C_VEL
LIN {X 0,Y 509.164,Z 480.772,A -85,B 0,C 180,E1 -5312.373,E2 -5312.373} C_VEL
LIN {X 0,Y 509.246,Z 477.918,A -85,B 0,C 180,E1 -5313.56,E2 -5313.56} C_VEL
LIN {X 0,Y 509.295,Z 475.322,A -85,B 0,C 180,E1 -5314.353,E2 -5314.353} C_VEL
LIN {X 0,Y 509.378,Z 470.206,A -85,B 0,C 180,E1 -5315.542,E2 -5315.542} C_VEL
LIN {X 0,Y 509.486,Z 465.179,A -85,B 0,C 180,E1 -5316.454,E2 -5316.454} C_VEL
LIN {X 0,Y 509.621,Z 457.799,A -85,B 0,C 180,E1 -5317.528,E2 -5317.528} C_VEL
LIN {X 0,Y 509.851,Z 448.852,A -85,B 0,C 180,E1 -5318.521,E2 -5318.521} C_VEL
LIN {X 0,Y 510.077,Z 441.085,A -85,B 0,C 180,E1 -5319.217,E2 -5319.217} C_VEL
LIN {X 0,Y 510.262,Z 432.898,A -85,B 0,C 180,E1 -5319.813,E2 -5319.813} C_VEL
LIN {X 0,Y 510.478,Z 424.359,A -85,B 0,C 180,E1 -5320.31,E2 -5320.31} C_VEL
LIN {X 0,Y 510.679,Z 413.089,A -85,B 0,C 180,E1 -5320.807,E2 -5320.807} C_VEL
LIN {X 0,Y 510.897,Z 401.531,A -85,B 0,C 180,E1 -5321.128,E2 -5321.128} C_VEL
LIN {X 0,Y 510.973,Z 377.997,A -85,B 0,C 180,E1 -5321.487,E2 -5321.487} C_VEL
LIN {X 0,Y 510.92,Z 332.434,A -85,B 0,C 180,E1 -5322.129,E2 -5322.129} C_VEL
LIN {X 0,Y 509.787,Z 324.133,A -85,B 0,C 180,E1 -5322.293,E2 -5322.293} C_VEL
LIN {X 0,Y 509.731,Z 323.526,A -85,B 0,C 180,E1 -5322.34,E2 -5322.34} C_VEL
LIN {X 0,Y 510.012,Z 307.971,A -85,B 0,C 180,E1 -5325.546,E2 -5325.546} C_VEL
LIN {X 0,Y 510.354,Z 294.108,A -85,B 0,C 180,E1 -5328.465,E2 -5328.465} C_VEL
LIN {X 0,Y 510.473,Z 286.298,A -85,B 0,C 180,E1 -5330.132,E2 -5330.132} C_VEL
LIN {X 0,Y 509.905,Z 281.885,A -85,B 0,C 180,E1 -5331.157,E2 -5331.157} C_VEL
LIN {X 0,Y 509.825,Z 281.789,A -85,B 0,C 180,E1 -5334.52,E2 -5334.52} C_VEL
LIN {X 0,Y 509.821,Z 281.789,A -85,B 0,C 180,E1 -5337.059,E2 -5337.059} C_VEL
LIN {X 0,Y 509.849,Z 281.789,A -85,B 0,C 180,E1 -5339.751,E2 -5339.751} C_VEL
LIN {X 0,Y 509.842,Z 281.785,A -85,B 0,C 180,E1 -5342.768,E2 -5342.768} C_VEL
LIN {X 0,Y 509.816,Z 281.794,A -85,B 0,C 180,E1 -5345.577,E2 -5345.577} C_VEL
LIN {X 0,Y 509.843,Z 281.784,A -85,B 0,C 180,E1 -5348.338,E2 -5348.338} C_VEL
LIN {X 0,Y 509.802,Z 281.795,A -85,B 0,C 180,E1 -5351.43,E2 -5351.43} C_VEL
LIN {X 0,Y 509.833,Z 281.788,A -85,B 0,C 180,E1 -5354.669,E2 -5354.669} C_VEL
LIN {X 0,Y 509.784,Z 281.795,A -85,B 0,C 180,E1 -5357.505,E2 -5357.505} C_VEL
LIN {X 0,Y 509.825,Z 281.79,A -85,B 0,C 180,E1 -5360.645,E2 -5360.645} C_VEL
LIN {X 0,Y 509.8,Z 281.79,A -85,B 0,C 180,E1 -5363.645,E2 -5363.645} C_VEL
LIN {X 0,Y 509.829,Z 281.79,A -85,B 0,C 180,E1 -5366.537,E2 -5366.537} C_VEL
LIN {X 0,Y 509.818,Z 281.789,A -85,B 0,C 180,E1 -5369.332,E2 -5369.332} C_VEL
LIN {X 0,Y 509.82,Z 281.788,A -85,B 0,C 180,E1 -5372.05,E2 -5372.05} C_VEL
LIN {X 0,Y 509.791,Z 281.799,A -85,B 0,C 180,E1 -5374.699,E2 -5374.699} C_VEL
LIN {X 0,Y 509.814,Z 281.788,A -85,B 0,C 180,E1 -5377.458,E2 -5377.458} C_VEL
LIN {X 0,Y 509.879,Z 281.781,A -85,B 0,C 180,E1 -5379.843,E2 -5379.843} C_VEL
LIN {X 0,Y 509.835,Z 281.792,A -85,B 0,C 180,E1 -5382.346,E2 -5382.346} C_VEL
LIN {X 0,Y 509.873,Z 281.784,A -85,B 0,C 180,E1 -5384.818,E2 -5384.818} C_VEL
LIN {X 0,Y 509.89,Z 281.784,A -85,B 0,C 180,E1 -5388.124,E2 -5388.124} C_VEL
LIN {X 0,Y 509.887,Z 281.779,A -85,B 0,C 180,E1 -5391.279,E2 -5391.279} C_VEL
LIN {X 0,Y 509.928,Z 281.778,A -85,B 0,C 180,E1 -5394.464,E2 -5394.464} C_VEL
LIN {X 0,Y 510.03,Z 281.764,A -85,B 0,C 180,E1 -5397.631,E2 -5397.631} C_VEL
LIN {X 0,Y 510.022,Z 281.771,A -85,B 0,C 180,E1 -5400,E2 -5400} C_VEL
LIN {X 0,Y 510.029,Z 281.764,A -85,B 0,C 180,E1 -5402.369,E2 -5402.369} C_VEL
LIN {X 0,Y 509.927,Z 281.778,A -85,B 0,C 180,E1 -5405.536,E2 -5405.536} C_VEL
LIN {X 0,Y 509.862,Z 281.789,A -85,B 0,C 180,E1 -5407.923,E2 -5407.923} C_VEL
LIN {X 0,Y 509.85,Z 281.785,A -85,B 0,C 180,E1 -5411.127,E2 -5411.127} C_VEL
LIN {X 0,Y 509.828,Z 281.793,A -85,B 0,C 180,E1 -5413.553,E2 -5413.553} C_VEL
LIN {X 0,Y 509.792,Z 281.794,A -85,B 0,C 180,E1 -5416.005,E2 -5416.005} C_VEL
LIN {X 0,Y 509.821,Z 281.787,A -85,B 0,C 180,E1 -5418.485,E2 -5418.485} C_VEL
LIN {X 0,Y 509.82,Z 281.789,A -85,B 0,C 180,E1 -5421.003,E2 -5421.003} C_VEL
LIN {X 0,Y 509.797,Z 281.797,A -85,B 0,C 180,E1 -5423.565,E2 -5423.565} C_VEL
LIN {X 0,Y 509.804,Z 281.789,A -85,B 0,C 180,E1 -5426.357,E2 -5426.357} C_VEL
LIN {X 0,Y 509.823,Z 281.79,A -85,B 0,C 180,E1 -5428.848,E2 -5428.848} C_VEL
LIN {X 0,Y 509.802,Z 281.793,A -85,B 0,C 180,E1 -5431.591,E2 -5431.591} C_VEL
LIN {X 0,Y 509.824,Z 281.787,A -85,B 0,C 180,E1 -5434.415,E2 -5434.415} C_VEL
LIN {X 0,Y 509.797,Z 281.795,A -85,B 0,C 180,E1 -5437.342,E2 -5437.342} C_VEL
LIN {X 0,Y 509.805,Z 281.79,A -85,B 0,C 180,E1 -5440.385,E2 -5440.385} C_VEL
LIN {X 0,Y 509.797,Z 281.791,A -85,B 0,C 180,E1 -5443.574,E2 -5443.574} C_VEL
LIN {X 0,Y 509.798,Z 281.793,A -85,B 0,C 180,E1 -5446.427,E2 -5446.427} C_VEL
LIN {X 0,Y 509.806,Z 281.789,A -85,B 0,C 180,E1 -5449.616,E2 -5449.616} C_VEL
LIN {X 0,Y 509.8,Z 281.798,A -85,B 0,C 180,E1 -5452.659,E2 -5452.659} C_VEL
LIN {X 0,Y 509.834,Z 281.786,A -85,B 0,C 180,E1 -5455.801,E2 -5455.801} C_VEL
LIN {X 0,Y 509.834,Z 281.792,A -85,B 0,C 180,E1 -5458.722,E2 -5458.722} C_VEL
LIN {X 0,Y 509.831,Z 281.787,A -85,B 0,C 180,E1 -5461.154,E2 -5461.154} C_VEL
LIN {X 0,Y 509.845,Z 281.786,A -85,B 0,C 180,E1 -5463.826,E2 -5463.826} C_VEL
LIN {X 0,Y 509.812,Z 281.784,A -85,B 0,C 180,E1 -5466.436,E2 -5466.436} C_VEL
LIN {X 0,Y 509.906,Z 281.995,A -85,B 0,C 180,E1 -5468.948,E2 -5468.948} C_VEL
LIN {X 0,Y 510.497,Z 288.043,A -85,B 0,C 180,E1 -5470.289,E2 -5470.289} C_VEL
LIN {X 0,Y 510.143,Z 301.706,A -85,B 0,C 180,E1 -5473.184,E2 -5473.184} C_VEL
LIN {X 0,Y 509.825,Z 315.37,A -85,B 0,C 180,E1 -5476.041,E2 -5476.041} C_VEL
LIN {X 0,Y 509.752,Z 323.665,A -85,B 0,C 180,E1 -5477.722,E2 -5477.722} C_VEL
LIN {X 0,Y 510.257,Z 327.434,A -85,B 0,C 180,E1 -5477.829,E2 -5477.829} C_VEL
LIN {X 0,Y 511.102,Z 335.147,A -85,B 0,C 180,E1 -5477.958,E2 -5477.958} C_VEL
LIN {X 0,Y 510.873,Z 399.253,A -85,B 0,C 180,E1 -5478.873,E2 -5478.873} C_VEL
LIN {X 0,Y 510.727,Z 408.418,A -85,B 0,C 180,E1 -5479.094,E2 -5479.094} C_VEL
LIN {X 0,Y 510.627,Z 416.888,A -85,B 0,C 180,E1 -5479.392,E2 -5479.392} C_VEL
LIN {X 0,Y 510.419,Z 425.391,A -85,B 0,C 180,E1 -5479.789,E2 -5479.789} C_VEL
LIN {X 0,Y 510.23,Z 433.724,A -85,B 0,C 180,E1 -5480.286,E2 -5480.286} C_VEL
LIN {X 0,Y 510.072,Z 441.761,A -85,B 0,C 180,E1 -5480.883,E2 -5480.883} C_VEL
LIN {X 0,Y 509.819,Z 450.433,A -85,B 0,C 180,E1 -5481.678,E2 -5481.678} C_VEL
LIN {X 0,Y 509.605,Z 458.939,A -85,B 0,C 180,E1 -5482.671,E2 -5482.671} C_VEL
LIN {X 0,Y 509.509,Z 465.61,A -85,B 0,C 180,E1 -5483.665,E2 -5483.665} C_VEL
LIN {X 0,Y 509.381,Z 469.989,A -85,B 0,C 180,E1 -5484.458,E2 -5484.458} C_VEL
LIN {X 0,Y 509.297,Z 475.15,A -85,B 0,C 180,E1 -5485.647,E2 -5485.647} C_VEL
LIN {X 0,Y 509.247,Z 477.787,A -85,B 0,C 180,E1 -5486.44,E2 -5486.44} C_VEL
LIN {X 0,Y 509.191,Z 480.68,A -85,B 0,C 180,E1 -5487.627,E2 -5487.627} C_VEL
LIN {X 0,Y 509.111,Z 481.928,A -85,B 0,C 180,E1 -5488.418,E2 -5488.418} C_VEL
LIN {X 0,Y 509.07,Z 482.706,A -85,B 0,C 180,E1 -5489.209,E2 -5489.209} C_VEL
LIN {X 0,Y 509.062,Z 483,A -85,B 0,C 180,E1 -5490,E2 -5490} C_VEL
LIN {X 0,Y 509.07,Z 482.705,A -85,B 0,C 180,E1 -5490.791,E2 -5490.791} C_VEL
LIN {X 0,Y 509.111,Z 481.927,A -85,B 0,C 180,E1 -5491.582,E2 -5491.582} C_VEL
LIN {X 0,Y 509.191,Z 480.679,A -85,B 0,C 180,E1 -5492.373,E2 -5492.373} C_VEL
LIN {X 0,Y 509.247,Z 477.786,A -85,B 0,C 180,E1 -5493.56,E2 -5493.56} C_VEL
LIN {X 0,Y 509.297,Z 475.149,A -85,B 0,C 180,E1 -5494.353,E2 -5494.353} C_VEL
LIN {X 0,Y 509.381,Z 469.986,A -85,B 0,C 180,E1 -5495.542,E2 -5495.542} C_VEL
LIN {X 0,Y 509.493,Z 464.854,A -85,B 0,C 180,E1 -5496.463,E2 -5496.463} C_VEL
LIN {X 0,Y 509.624,Z 457.436,A -85,B 0,C 180,E1 -5497.528,E2 -5497.528} C_VEL
LIN {X 0,Y 509.83,Z 449.419,A -85,B 0,C 180,E1 -5498.422,E2 -5498.422} C_VEL
LIN {X 0,Y 510.072,Z 441.765,A -85,B 0,C 180,E1 -5499.117,E2 -5499.117} C_VEL
LIN {X 0,Y 510.23,Z 433.725,A -85,B 0,C 180,E1 -5499.714,E2 -5499.714} C_VEL
LIN {X 0,Y 510.419,Z 425.393,A -85,B 0,C 180,E1 -5500.211,E2 -5500.211} C_VEL
LIN {X 0,Y 510.626,Z 416.891,A -85,B 0,C 180,E1 -5500.608,E2 -5500.608} C_VEL
LIN {X 0,Y 510.741,Z 406.758,A -85,B 0,C 180,E1 -5500.956,E2 -5500.956} C_VEL
LIN {X 0,Y 510.906,Z 393.983,A -85,B 0,C 180,E1 -5501.219,E2 -5501.219} C_VEL
LIN {X 0,Y 511.014,Z 333.178,A -85,B 0,C 180,E1 -5502.071,E2 -5502.071} C_VEL
LIN {X 0,Y 509.783,Z 323.972,A -85,B 0,C 180,E1 -5502.252,E2 -5502.252} C_VEL
LIN {X 0,Y 509.755,Z 321.226,A -85,B 0,C 180,E1 -5502.744,E2 -5502.744} C_VEL
LIN {X 0,Y 510.029,Z 306.684,A -85,B 0,C 180,E1 -5505.771,E2 -5505.771} C_VEL
LIN {X 0,Y 510.424,Z 291.946,A -85,B 0,C 180,E1 -5508.878,E2 -5508.878} C_VEL
LIN {X 0,Y 510.293,Z 284.305,A -85,B 0,C 180,E1 -5510.524,E2 -5510.524} C_VEL
LIN {X 0,Y 509.867,Z 281.894,A -85,B 0,C 180,E1 -5511.106,E2 -5511.106} C_VEL
LIN {X 0,Y 509.832,Z 281.788,A -85,B 0,C 180,E1 -5514.427,E2 -5514.427} C_VEL
LIN {X 0,Y 509.819,Z 281.789,A -85,B 0,C 180,E1 -5517.059,E2 -5517.059} C_VEL
LIN {X 0,Y 509.847,Z 281.789,A -85,B 0,C 180,E1 -5519.751,E2 -5519.751} C_VEL
LIN {X 0,Y 509.839,Z 281.786,A -85,B 0,C 180,E1 -5522.768,E2 -5522.768} C_VEL
LIN {X 0,Y 509.808,Z 281.794,A -85,B 0,C 180,E1 -5525.576,E2 -5525.576} C_VEL
LIN {X 0,Y 509.842,Z 281.784,A -85,B 0,C 180,E1 -5528.338,E2 -5528.338} C_VEL
LIN {X 0,Y 509.8,Z 281.795,A -85,B 0,C 180,E1 -5531.43,E2 -5531.43} C_VEL
LIN {X 0,Y 509.832,Z 281.788,A -85,B 0,C 180,E1 -5534.669,E2 -5534.669} C_VEL
LIN {X 0,Y 509.783,Z 281.795,A -85,B 0,C 180,E1 -5537.505,E2 -5537.505} C_VEL
LIN {X 0,Y 509.824,Z 281.791,A -85,B 0,C 180,E1 -5540.646,E2 -5540.646} C_VEL
LIN {X 0,Y 509.794,Z 281.791,A -85,B 0,C 180,E1 -5543.644,E2 -5543.644} C_VEL
LIN {X 0,Y 509.829,Z 281.79,A -85,B 0,C 180,E1 -5546.537,E2 -5546.537} C_VEL
LIN {X 0,Y 509.818,Z 281.789,A -85,B 0,C 180,E1 -5549.332,E2 -5549.332} C_VEL
LIN {X 0,Y 509.819,Z 281.788,A -85,B 0,C 180,E1 -5552.05,E2 -5552.05} C_VEL
LIN {X 0,Y 509.791,Z 281.799,A -85,B 0,C 180,E1 -5554.699,E2 -5554.699} C_VEL
LIN {X 0,Y 509.813,Z 281.788,A -85,B 0,C 180,E1 -5557.459,E2 -5557.459} C_VEL
LIN {X 0,Y 509.878,Z 281.781,A -85,B 0,C 180,E1 -5559.843,E2 -5559.843} C_VEL
LIN {X 0,Y 509.834,Z 281.793,A -85,B 0,C 180,E1 -5562.346,E2 -5562.346} C_VEL
LIN {X 0,Y 509.873,Z 281.784,A -85,B 0,C 180,E1 -5564.818,E2 -5564.818} C_VEL
LIN {X 0,Y 509.89,Z 281.784,A -85,B 0,C 180,E1 -5568.124,E2 -5568.124} C_VEL
LIN {X 0,Y 509.871,Z 281.781,A -85,B 0,C 180,E1 -5571.279,E2 -5571.279} C_VEL
LIN {X 0,Y 509.928,Z 281.778,A -85,B 0,C 180,E1 -5574.464,E2 -5574.464} C_VEL
LIN {X 0,Y 510.03,Z 281.764,A -85,B 0,C 180,E1 -5577.631,E2 -5577.631} C_VEL
LIN {X 0,Y 510.022,Z 281.771,A -85,B 0,C 180,E1 -5580,E2 -5580} C_VEL
LIN {X 0,Y 510.03,Z 281.764,A -85,B 0,C 180,E1 -5582.369,E2 -5582.369} C_VEL
LIN {X 0,Y 509.928,Z 281.778,A -85,B 0,C 180,E1 -5585.536,E2 -5585.536} C_VEL
LIN {X 0,Y 509.862,Z 281.789,A -85,B 0,C 180,E1 -5587.923,E2 -5587.923} C_VEL
LIN {X 0,Y 509.849,Z 281.785,A -85,B 0,C 180,E1 -5591.127,E2 -5591.127} C_VEL
LIN {X 0,Y 509.812,Z 281.795,A -85,B 0,C 180,E1 -5593.554,E2 -5593.554} C_VEL
LIN {X 0,Y 509.791,Z 281.794,A -85,B 0,C 180,E1 -5596.005,E2 -5596.005} C_VEL
LIN {X 0,Y 509.821,Z 281.787,A -85,B 0,C 180,E1 -5598.485,E2 -5598.485} C_VEL
LIN {X 0,Y 509.821,Z 281.789,A -85,B 0,C 180,E1 -5601.003,E2 -5601.003} C_VEL
LIN {X 0,Y 509.798,Z 281.797,A -85,B 0,C 180,E1 -5603.565,E2 -5603.565} C_VEL
LIN {X 0,Y 509.804,Z 281.789,A -85,B 0,C 180,E1 -5606.357,E2 -5606.357} C_VEL
LIN {X 0,Y 509.82,Z 281.79,A -85,B 0,C 180,E1 -5608.848,E2 -5608.848} C_VEL
LIN {X 0,Y 509.788,Z 281.795,A -85,B 0,C 180,E1 -5611.593,E2 -5611.593} C_VEL
LIN {X 0,Y 509.824,Z 281.787,A -85,B 0,C 180,E1 -5614.416,E2 -5614.416} C_VEL
LIN {X 0,Y 509.797,Z 281.795,A -85,B 0,C 180,E1 -5617.343,E2 -5617.343} C_VEL
LIN {X 0,Y 509.806,Z 281.79,A -85,B 0,C 180,E1 -5620.385,E2 -5620.385} C_VEL
LIN {X 0,Y 509.798,Z 281.791,A -85,B 0,C 180,E1 -5623.574,E2 -5623.574} C_VEL
LIN {X 0,Y 509.799,Z 281.792,A -85,B 0,C 180,E1 -5626.427,E2 -5626.427} C_VEL
LIN {X 0,Y 509.807,Z 281.789,A -85,B 0,C 180,E1 -5629.616,E2 -5629.616} C_VEL
LIN {X 0,Y 509.801,Z 281.797,A -85,B 0,C 180,E1 -5632.659,E2 -5632.659} C_VEL
LIN {X 0,Y 509.796,Z 281.79,A -85,B 0,C 180,E1 -5633.694,E2 -5633.694} C_VEL
LIN {X 0,Y 509.129,Z 281.879,A -85,B 0,C 180,E1 -5634.354,E2 -5634.354} C_VEL
LIN {X 0,Y 506.31,Z 282.23,A -85,B 0,C 180,E1 -5635.426,E2 -5635.426} C_VEL
LIN {X 0,Y 503.921,Z 282.528,A -85,B 0,C 180,E1 -5636.29,E2 -5636.29} C_VEL
LIN {X 0,Y 502.878,Z 282.657,A -85,B 0,C 180,E1 -5636.956,E2 -5636.956} C_VEL
LIN {X 0,Y 502.784,Z 282.665,A -85,B 0,C 180,E1 -5637.182,E2 -5637.182} C_VEL
LIN {X 0,Y 502.761,Z 282.669,A -85,B 0,C 180,E1 -5640.076,E2 -5640.076} C_VEL
LIN {X 0,Y 502.772,Z 282.674,A -85,B 0,C 180,E1 -5642.53,E2 -5642.53} C_VEL
LIN {X 0,Y 502.769,Z 282.668,A -85,B 0,C 180,E1 -5645.314,E2 -5645.314} C_VEL
LIN {X 0,Y 502.771,Z 282.651,A -85,B 0,C 180,E1 -5647.827,E2 -5647.827} C_VEL
LIN {X 0,Y 502.833,Z 282.887,A -85,B 0,C 180,E1 -5648.881,E2 -5648.881} C_VEL
LIN {X 0,Y 503.451,Z 287.836,A -85,B 0,C 180,E1 -5650.001,E2 -5650.001} C_VEL
LIN {X 0,Y 503.231,Z 299.545,A -85,B 0,C 180,E1 -5652.527,E2 -5652.527} C_VEL
LIN {X 0,Y 502.885,Z 313.206,A -85,B 0,C 180,E1 -5655.431,E2 -5655.431} C_VEL
LIN {X 0,Y 502.697,Z 323.755,A -85,B 0,C 180,E1 -5657.599,E2 -5657.599} C_VEL
LIN {X 0,Y 503.458,Z 329.121,A -85,B 0,C 180,E1 -5657.732,E2 -5657.732} C_VEL
LIN {X 0,Y 504.197,Z 335.343,A -85,B 0,C 180,E1 -5657.839,E2 -5657.839} C_VEL
LIN {X 0,Y 503.945,Z 399.455,A -85,B 0,C 180,E1 -5658.767,E2 -5658.767} C_VEL
LIN {X 0,Y 503.786,Z 408.613,A -85,B 0,C 180,E1 -5658.992,E2 -5658.992} C_VEL
LIN {X 0,Y 503.605,Z 418.24,A -85,B 0,C 180,E1 -5659.344,E2 -5659.344} C_VEL
LIN {X 0,Y 503.451,Z 428.308,A -85,B 0,C 180,E1 -5659.849,E2 -5659.849} C_VEL
LIN {X 0,Y 503.137,Z 438.759,A -85,B 0,C 180,E1 -5660.554,E2 -5660.554} C_VEL
LIN {X 0,Y 502.871,Z 446.924,A -85,B 0,C 180,E1 -5661.258,E2 -5661.258} C_VEL
LIN {X 0,Y 502.685,Z 453.661,A -85,B 0,C 180,E1 -5661.963,E2 -5661.963} C_VEL
LIN {X 0,Y 502.547,Z 460.039,A -85,B 0,C 180,E1 -5662.77,E2 -5662.77} C_VEL
LIN {X 0,Y 502.453,Z 465.343,A -85,B 0,C 180,E1 -5663.575,E2 -5663.575} C_VEL
LIN {X 0,Y 502.315,Z 469.772,A -85,B 0,C 180,E1 -5664.38,E2 -5664.38} C_VEL
LIN {X 0,Y 502.154,Z 473.463,A -85,B 0,C 180,E1 -5665.183,E2 -5665.183} C_VEL
LIN {X 0,Y 502.203,Z 476.474,A -85,B 0,C 180,E1 -5665.988,E2 -5665.988} C_VEL
LIN {X 0,Y 502.135,Z 478.808,A -85,B 0,C 180,E1 -5666.791,E2 -5666.791} C_VEL
LIN {X 0,Y 502.094,Z 480.588,A -85,B 0,C 180,E1 -5667.593,E2 -5667.593} C_VEL
LIN {X 0,Y 502.035,Z 481.873,A -85,B 0,C 180,E1 -5668.396,E2 -5668.396} C_VEL
LIN {X 0,Y 501.987,Z 482.687,A -85,B 0,C 180,E1 -5669.198,E2 -5669.198} C_VEL
LIN {X 0,Y 501.978,Z 482.997,A -85,B 0,C 180,E1 -5670,E2 -5670} C_VEL
LIN {X 0,Y 501.988,Z 482.724,A -85,B 0,C 180,E1 -5670.802,E2 -5670.802} C_VEL
LIN {X 0,Y 502.035,Z 481.982,A -85,B 0,C 180,E1 -5671.604,E2 -5671.604} C_VEL
LIN {X 0,Y 502.069,Z 480.771,A -85,B 0,C 180,E1 -5672.407,E2 -5672.407} C_VEL
LIN {X 0,Y 502.171,Z 477.916,A -85,B 0,C 180,E1 -5673.611,E2 -5673.611} C_VEL
LIN {X 0,Y 502.188,Z 475.319,A -85,B 0,C 180,E1 -5674.414,E2 -5674.414} C_VEL
LIN {X 0,Y 502.325,Z 470.203,A -85,B 0,C 180,E1 -5675.62,E2 -5675.62} C_VEL
LIN {X 0,Y 502.424,Z 464.251,A -85,B 0,C 180,E1 -5676.704,E2 -5676.704} C_VEL
LIN {X 0,Y 502.598,Z 456.117,A -85,B 0,C 180,E1 -5677.836,E2 -5677.836} C_VEL
LIN {X 0,Y 502.811,Z 448.845,A -85,B 0,C 180,E1 -5678.642,E2 -5678.642} C_VEL
LIN {X 0,Y 503.059,Z 441.077,A -85,B 0,C 180,E1 -5679.346,E2 -5679.346} C_VEL
LIN {X 0,Y 503.259,Z 432.888,A -85,B 0,C 180,E1 -5679.951,E2 -5679.951} C_VEL
LIN {X 0,Y 503.487,Z 424.347,A -85,B 0,C 180,E1 -5680.455,E2 -5680.455} C_VEL
LIN {X 0,Y 503.72,Z 413.071,A -85,B 0,C 180,E1 -5680.958,E2 -5680.958} C_VEL
LIN {X 0,Y 503.937,Z 401.556,A -85,B 0,C 180,E1 -5681.282,E2 -5681.282} C_VEL
LIN {X 0,Y 504.016,Z 377.604,A -85,B 0,C 180,E1 -5681.653,E2 -5681.653} C_VEL
LIN {X 0,Y 503.985,Z 333.265,A -85,B 0,C 180,E1 -5682.286,E2 -5682.286} C_VEL
LIN {X 0,Y 502.73,Z 324.118,A -85,B 0,C 180,E1 -5682.468,E2 -5682.468} C_VEL
LIN {X 0,Y 502.678,Z 323.522,A -85,B 0,C 180,E1 -5682.516,E2 -5682.516} C_VEL
LIN {X 0,Y 502.936,Z 309.725,A -85,B 0,C 180,E1 -5685.397,E2 -5685.397} C_VEL
LIN {X 0,Y 503.337,Z 295.437,A -85,B 0,C 180,E1 -5688.444,E2 -5688.444} C_VEL
LIN {X 0,Y 503.367,Z 286.296,A -85,B 0,C 180,E1 -5690.429,E2 -5690.429} C_VEL
LIN {X 0,Y 502.851,Z 282.773,A -85,B 0,C 180,E1 -5691.261,E2 -5691.261} C_VEL
LIN {X 0,Y 502.765,Z 282.666,A -85,B 0,C 180,E1 -5693.914,E2 -5693.914} C_VEL
LIN {X 0,Y 502.782,Z 282.664,A -85,B 0,C 180,E1 -5696.57,E2 -5696.57} C_VEL
LIN {X 0,Y 502.808,Z 282.664,A -85,B 0,C 180,E1 -5699.933,E2 -5699.933} C_VEL
LIN {X 0,Y 502.799,Z 282.665,A -85,B 0,C 180,E1 -5703.033,E2 -5703.033} C_VEL
LIN {X 0,Y 502.762,Z 282.668,A -85,B 0,C 180,E1 -5705.951,E2 -5705.951} C_VEL
LIN {X 0,Y 502.79,Z 282.667,A -85,B 0,C 180,E1 -5708.976,E2 -5708.976} C_VEL
LIN {X 0,Y 502.739,Z 282.669,A -85,B 0,C 180,E1 -5712.191,E2 -5712.191} C_VEL
LIN {X 0,Y 502.779,Z 282.668,A -85,B 0,C 180,E1 -5715.469,E2 -5715.469} C_VEL
LIN {X 0,Y 502.757,Z 282.674,A -85,B 0,C 180,E1 -5718.928,E2 -5718.928} C_VEL
LIN {X 0,Y 502.782,Z 282.664,A -85,B 0,C 180,E1 -5722.045,E2 -5722.045} C_VEL
LIN {X 0,Y 502.782,Z 282.671,A -85,B 0,C 180,E1 -5725.033,E2 -5725.033} C_VEL
LIN {X 0,Y 502.769,Z 282.666,A -85,B 0,C 180,E1 -5727.914,E2 -5727.914} C_VEL
LIN {X 0,Y 502.794,Z 282.671,A -85,B 0,C 180,E1 -5730.71,E2 -5730.71} C_VEL
LIN {X 0,Y 502.765,Z 282.667,A -85,B 0,C 180,E1 -5733.459,E2 -5733.459} C_VEL
LIN {X 0,Y 502.754,Z 282.669,A -85,B 0,C 180,E1 -5736.084,E2 -5736.084} C_VEL
LIN {X 0,Y 502.82,Z 282.659,A -85,B 0,C 180,E1 -5739.463,E2 -5739.463} C_VEL
LIN {X 0,Y 502.773,Z 282.668,A -85,B 0,C 180,E1 -5742.09,E2 -5742.09} C_VEL
LIN {X 0,Y 502.814,Z 282.66,A -85,B 0,C 180,E1 -5745.428,E2 -5745.428} C_VEL
LIN {X 0,Y 502.864,Z 282.657,A -85,B 0,C 180,E1 -5748.716,E2 -5748.716} C_VEL
LIN {X 0,Y 502.859,Z 282.659,A -85,B 0,C 180,E1 -5751.966,E2 -5751.966} C_VEL
LIN {X 0,Y 502.885,Z 282.657,A -85,B 0,C 180,E1 -5754.386,E2 -5754.386} C_VEL
LIN {X 0,Y 502.997,Z 282.639,A -85,B 0,C 180,E1 -5757.598,E2 -5757.598} C_VEL
LIN {X 0,Y 502.991,Z 282.647,A -85,B 0,C 180,E1 -5760,E2 -5760} C_VEL
LIN {X 0,Y 502.997,Z 282.64,A -85,B 0,C 180,E1 -5762.402,E2 -5762.402} C_VEL
LIN {X 0,Y 502.884,Z 282.656,A -85,B 0,C 180,E1 -5765.614,E2 -5765.614} C_VEL
LIN {X 0,Y 502.834,Z 282.663,A -85,B 0,C 180,E1 -5768.034,E2 -5768.034} C_VEL
LIN {X 0,Y 502.825,Z 282.661,A -85,B 0,C 180,E1 -5771.284,E2 -5771.284} C_VEL
LIN {X 0,Y 502.813,Z 282.66,A -85,B 0,C 180,E1 -5774.572,E2 -5774.572} C_VEL
LIN {X 0,Y 502.773,Z 282.669,A -85,B 0,C 180,E1 -5777.91,E2 -5777.91} C_VEL
LIN {X 0,Y 502.791,Z 282.663,A -85,B 0,C 180,E1 -5780.528,E2 -5780.528} C_VEL
LIN {X 0,Y 502.77,Z 282.669,A -85,B 0,C 180,E1 -5783.042,E2 -5783.042} C_VEL
LIN {X 0,Y 502.765,Z 282.67,A -85,B 0,C 180,E1 -5785.68,E2 -5785.68} C_VEL
LIN {X 0,Y 502.759,Z 282.667,A -85,B 0,C 180,E1 -5788.378,E2 -5788.378} C_VEL
LIN {X 0,Y 502.776,Z 282.672,A -85,B 0,C 180,E1 -5791.145,E2 -5791.145} C_VEL
LIN {X 0,Y 502.776,Z 282.665,A -85,B 0,C 180,E1 -5793.996,E2 -5793.996} C_VEL
LIN {X 0,Y 502.754,Z 282.675,A -85,B 0,C 180,E1 -5797.176,E2 -5797.176} C_VEL
LIN {X 0,Y 502.762,Z 282.666,A -85,B 0,C 180,E1 -5800.018,E2 -5800.018} C_VEL
LIN {X 0,Y 502.739,Z 282.674,A -85,B 0,C 180,E1 -5803.235,E2 -5803.235} C_VEL
LIN {X 0,Y 502.771,Z 282.666,A -85,B 0,C 180,E1 -5805.66,E2 -5805.66} C_VEL
LIN {X 0,Y 502.757,Z 282.673,A -85,B 0,C 180,E1 -5809.013,E2 -5809.013} C_VEL
LIN {X 0,Y 502.765,Z 282.667,A -85,B 0,C 180,E1 -5812.045,E2 -5812.045} C_VEL
LIN {X 0,Y 502.783,Z 282.667,A -85,B 0,C 180,E1 -5815.034,E2 -5815.034} C_VEL
LIN {X 0,Y 502.774,Z 282.666,A -85,B 0,C 180,E1 -5817.916,E2 -5817.916} C_VEL
LIN {X 0,Y 502.799,Z 282.667,A -85,B 0,C 180,E1 -5820.711,E2 -5820.711} C_VEL
LIN {X 0,Y 502.77,Z 282.665,A -85,B 0,C 180,E1 -5823.46,E2 -5823.46} C_VEL
LIN {X 0,Y 502.762,Z 282.668,A -85,B 0,C 180,E1 -5826.085,E2 -5826.085} C_VEL
LIN {X 0,Y 502.878,Z 282.872,A -85,B 0,C 180,E1 -5828.833,E2 -5828.833} C_VEL
LIN {X 0,Y 503.483,Z 288.044,A -85,B 0,C 180,E1 -5830.002,E2 -5830.002} C_VEL
LIN {X 0,Y 503.228,Z 299.755,A -85,B 0,C 180,E1 -5832.527,E2 -5832.527} C_VEL
LIN {X 0,Y 502.883,Z 313.418,A -85,B 0,C 180,E1 -5835.431,E2 -5835.431} C_VEL
LIN {X 0,Y 502.717,Z 323.529,A -85,B 0,C 180,E1 -5837.531,E2 -5837.531} C_VEL
LIN {X 0,Y 502.901,Z 325.318,A -85,B 0,C 180,E1 -5837.615,E2 -5837.615} C_VEL
LIN {X 0,Y 504.16,Z 336.027,A -85,B 0,C 180,E1 -5837.803,E2 -5837.803} C_VEL
LIN {X 0,Y 503.917,Z 399.307,A -85,B 0,C 180,E1 -5838.718,E2 -5838.718} C_VEL
LIN {X 0,Y 503.774,Z 408.418,A -85,B 0,C 180,E1 -5838.941,E2 -5838.941} C_VEL
LIN {X 0,Y 503.663,Z 416.888,A -85,B 0,C 180,E1 -5839.244,E2 -5839.244} C_VEL
LIN {X 0,Y 503.435,Z 425.391,A -85,B 0,C 180,E1 -5839.646,E2 -5839.646} C_VEL
LIN {X 0,Y 503.239,Z 433.724,A -85,B 0,C 180,E1 -5840.15,E2 -5840.15} C_VEL
LIN {X 0,Y 503.046,Z 441.761,A -85,B 0,C 180,E1 -5840.755,E2 -5840.755} C_VEL
LIN {X 0,Y 502.771,Z 450.433,A -85,B 0,C 180,E1 -5841.56,E2 -5841.56} C_VEL
LIN {X 0,Y 502.543,Z 458.939,A -85,B 0,C 180,E1 -5842.568,E2 -5842.568} C_VEL
LIN {X 0,Y 502.436,Z 465.61,A -85,B 0,C 180,E1 -5843.575,E2 -5843.575} C_VEL
LIN {X 0,Y 502.33,Z 469.989,A -85,B 0,C 180,E1 -5844.38,E2 -5844.38} C_VEL
LIN {X 0,Y 502.189,Z 475.15,A -85,B 0,C 180,E1 -5845.586,E2 -5845.586} C_VEL
LIN {X 0,Y 502.171,Z 477.787,A -85,B 0,C 180,E1 -5846.389,E2 -5846.389} C_VEL
LIN {X 0,Y 502.093,Z 480.68,A -85,B 0,C 180,E1 -5847.593,E2 -5847.593} C_VEL
LIN {X 0,Y 502.035,Z 481.928,A -85,B 0,C 180,E1 -5848.396,E2 -5848.396} C_VEL
LIN {X 0,Y 501.987,Z 482.706,A -85,B 0,C 180,E1 -5849.198,E2 -5849.198} C_VEL
LIN {X 0,Y 501.977,Z 483,A -85,B 0,C 180,E1 -5850,E2 -5850} C_VEL
LIN {X 0,Y 501.987,Z 482.705,A -85,B 0,C 180,E1 -5850.802,E2 -5850.802} C_VEL
LIN {X 0,Y 502.035,Z 481.927,A -85,B 0,C 180,E1 -5851.604,E2 -5851.604} C_VEL
LIN {X 0,Y 502.093,Z 480.679,A -85,B 0,C 180,E1 -5852.407,E2 -5852.407} C_VEL
LIN {X 0,Y 502.171,Z 477.786,A -85,B 0,C 180,E1 -5853.611,E2 -5853.611} C_VEL
LIN {X 0,Y 502.189,Z 475.149,A -85,B 0,C 180,E1 -5854.414,E2 -5854.414} C_VEL
LIN {X 0,Y 502.33,Z 469.986,A -85,B 0,C 180,E1 -5855.62,E2 -5855.62} C_VEL
LIN {X 0,Y 502.43,Z 463.934,A -85,B 0,C 180,E1 -5856.711,E2 -5856.711} C_VEL
LIN {X 0,Y 502.564,Z 457.436,A -85,B 0,C 180,E1 -5857.634,E2 -5857.634} C_VEL
LIN {X 0,Y 502.789,Z 449.419,A -85,B 0,C 180,E1 -5858.541,E2 -5858.541} C_VEL
LIN {X 0,Y 503.046,Z 441.765,A -85,B 0,C 180,E1 -5859.245,E2 -5859.245} C_VEL
LIN {X 0,Y 503.239,Z 433.725,A -85,B 0,C 180,E1 -5859.85,E2 -5859.85} C_VEL
LIN {X 0,Y 503.435,Z 425.393,A -85,B 0,C 180,E1 -5860.354,E2 -5860.354} C_VEL
LIN {X 0,Y 503.663,Z 416.891,A -85,B 0,C 180,E1 -5860.756,E2 -5860.756} C_VEL
LIN {X 0,Y 503.78,Z 406.758,A -85,B 0,C 180,E1 -5861.11,E2 -5861.11} C_VEL
LIN {X 0,Y 503.96,Z 394.374,A -85,B 0,C 180,E1 -5861.37,E2 -5861.37} C_VEL
LIN {X 0,Y 504.001,Z 333.178,A -85,B 0,C 180,E1 -5862.242,E2 -5862.242} C_VEL
LIN {X 0,Y 502.746,Z 324.078,A -85,B 0,C 180,E1 -5862.421,E2 -5862.421} C_VEL
LIN {X 0,Y 502.715,Z 323.036,A -85,B 0,C 180,E1 -5862.556,E2 -5862.556} C_VEL
LIN {X 0,Y 503.009,Z 307.562,A -85,B 0,C 180,E1 -5865.81,E2 -5865.81} C_VEL
LIN {X 0,Y 503.389,Z 293.897,A -85,B 0,C 180,E1 -5868.73,E2 -5868.73} C_VEL
LIN {X 0,Y 503.354,Z 286.088,A -85,B 0,C 180,E1 -5870.429,E2 -5870.429} C_VEL
LIN {X 0,Y 502.85,Z 282.773,A -85,B 0,C 180,E1 -5871.215,E2 -5871.215} C_VEL
LIN {X 0,Y 502.762,Z 282.668,A -85,B 0,C 180,E1 -5873.915,E2 -5873.915} C_VEL
LIN {X 0,Y 502.78,Z 282.664,A -85,B 0,C 180,E1 -5876.57,E2 -5876.57} C_VEL
LIN {X 0,Y 502.805,Z 282.664,A -85,B 0,C 180,E1 -5879.933,E2 -5879.933} C_VEL
LIN {X 0,Y 502.797,Z 282.665,A -85,B 0,C 180,E1 -5883.033,E2 -5883.033} C_VEL
LIN {X 0,Y 502.757,Z 282.668,A -85,B 0,C 180,E1 -5885.951,E2 -5885.951} C_VEL
LIN {X 0,Y 502.788,Z 282.668,A -85,B 0,C 180,E1 -5888.976,E2 -5888.976} C_VEL
LIN {X 0,Y 502.738,Z 282.669,A -85,B 0,C 180,E1 -5892.191,E2 -5892.191} C_VEL
LIN {X 0,Y 502.778,Z 282.668,A -85,B 0,C 180,E1 -5895.47,E2 -5895.47} C_VEL
LIN {X 0,Y 502.756,Z 282.674,A -85,B 0,C 180,E1 -5898.928,E2 -5898.928} C_VEL
LIN {X 0,Y 502.78,Z 282.664,A -85,B 0,C 180,E1 -5902.045,E2 -5902.045} C_VEL
LIN {X 0,Y 502.779,Z 282.671,A -85,B 0,C 180,E1 -5905.033,E2 -5905.033} C_VEL
LIN {X 0,Y 502.768,Z 282.666,A -85,B 0,C 180,E1 -5907.914,E2 -5907.914} C_VEL
LIN {X 0,Y 502.793,Z 282.671,A -85,B 0,C 180,E1 -5910.71,E2 -5910.71} C_VEL
LIN {X 0,Y 502.764,Z 282.666,A -85,B 0,C 180,E1 -5913.459,E2 -5913.459} C_VEL
LIN {X 0,Y 502.753,Z 282.669,A -85,B 0,C 180,E1 -5916.084,E2 -5916.084} C_VEL
LIN {X 0,Y 502.819,Z 282.659,A -85,B 0,C 180,E1 -5919.464,E2 -5919.464} C_VEL
LIN {X 0,Y 502.772,Z 282.669,A -85,B 0,C 180,E1 -5922.09,E2 -5922.09} C_VEL
LIN {X 0,Y 502.813,Z 282.66,A -85,B 0,C 180,E1 -5925.428,E2 -5925.428} C_VEL
LIN {X 0,Y 502.864,Z 282.657,A -85,B 0,C 180,E1 -5928.717,E2 -5928.717} C_VEL
LIN {X 0,Y 502.837,Z 282.662,A -85,B 0,C 180,E1 -5931.966,E2 -5931.966} C_VEL
LIN {X 0,Y 502.885,Z 282.656,A -85,B 0,C 180,E1 -5934.386,E2 -5934.386} C_VEL
LIN {X 0,Y 502.997,Z 282.639,A -85,B 0,C 180,E1 -5937.598,E2 -5937.598} C_VEL
LIN {X 0,Y 502.991,Z 282.647,A -85,B 0,C 180,E1 -5940,E2 -5940} C_VEL
LIN {X 0,Y 502.997,Z 282.64,A -85,B 0,C 180,E1 -5942.402,E2 -5942.402} C_VEL
LIN {X 0,Y 502.884,Z 282.656,A -85,B 0,C 180,E1 -5945.614,E2 -5945.614} C_VEL
LIN {X 0,Y 502.834,Z 282.663,A -85,B 0,C 180,E1 -5948.035,E2 -5948.035} C_VEL
LIN {X 0,Y 502.825,Z 282.661,A -85,B 0,C 180,E1 -5951.284,E2 -5951.284} C_VEL
LIN {X 0,Y 502.812,Z 282.66,A -85,B 0,C 180,E1 -5954.572,E2 -5954.572} C_VEL
LIN {X 0,Y 502.773,Z 282.669,A -85,B 0,C 180,E1 -5957.91,E2 -5957.91} C_VEL
LIN {X 0,Y 502.792,Z 282.663,A -85,B 0,C 180,E1 -5960.528,E2 -5960.528} C_VEL
LIN {X 0,Y 502.771,Z 282.668,A -85,B 0,C 180,E1 -5963.042,E2 -5963.042} C_VEL
LIN {X 0,Y 502.766,Z 282.671,A -85,B 0,C 180,E1 -5965.68,E2 -5965.68} C_VEL
LIN {X 0,Y 502.759,Z 282.667,A -85,B 0,C 180,E1 -5968.378,E2 -5968.378} C_VEL
LIN {X 0,Y 502.756,Z 282.674,A -85,B 0,C 180,E1 -5971.146,E2 -5971.146} C_VEL
LIN {X 0,Y 502.776,Z 282.665,A -85,B 0,C 180,E1 -5973.996,E2 -5973.996} C_VEL
LIN {X 0,Y 502.754,Z 282.675,A -85,B 0,C 180,E1 -5977.176,E2 -5977.176} C_VEL
LIN {X 0,Y 502.763,Z 282.666,A -85,B 0,C 180,E1 -5980.018,E2 -5980.018} C_VEL
LIN {X 0,Y 502.74,Z 282.674,A -85,B 0,C 180,E1 -5983.235,E2 -5983.235} C_VEL
LIN {X 0,Y 502.772,Z 282.666,A -85,B 0,C 180,E1 -5985.661,E2 -5985.661} C_VEL
LIN {X 0,Y 502.757,Z 282.673,A -85,B 0,C 180,E1 -5989.013,E2 -5989.013} C_VEL
LIN {X 0,Y 502.766,Z 282.667,A -85,B 0,C 180,E1 -5992.045,E2 -5992.045} C_VEL
LIN {X 0,Y 502.784,Z 282.667,A -85,B 0,C 180,E1 -5995.034,E2 -5995.034} C_VEL
LIN {X 0,Y 502.784,Z 282.665,A -85,B 0,C 180,E1 -5997.182,E2 -5997.182} C_VEL
LIN {X 0,Y 502.089,Z 282.751,A -85,B 0,C 180,E1 -5997.85,E2 -5997.85} C_VEL
LIN {X 0,Y 499.216,Z 283.112,A -85,B 0,C 180,E1 -5998.936,E2 -5998.936} C_VEL
LIN {X 0,Y 496.802,Z 283.412,A -85,B 0,C 180,E1 -5999.81,E2 -5999.81} C_VEL
LIN {X 0,Y 495.768,Z 283.546,A -85,B 0,C 180,E1 -6000.486,E2 -6000.486} C_VEL
LIN {X 0,Y 495.684,Z 283.549,A -85,B 0,C 180,E1 -6000.715,E2 -6000.715} C_VEL
LIN {X 0,Y 495.737,Z 283.542,A -85,B 0,C 180,E1 -6003.271,E2 -6003.271} C_VEL
LIN {X 0,Y 495.708,Z 283.548,A -85,B 0,C 180,E1 -6005.723,E2 -6005.723} C_VEL
LIN {X 0,Y 495.802,Z 283.747,A -85,B 0,C 180,E1 -6008.756,E2 -6008.756} C_VEL
LIN {X 0,Y 496.456,Z 289.79,A -85,B 0,C 180,E1 -6010.139,E2 -6010.139} C_VEL
LIN {X 0,Y 496.158,Z 301.499,A -85,B 0,C 180,E1 -6012.695,E2 -6012.695} C_VEL
LIN {X 0,Y 495.819,Z 315.16,A -85,B 0,C 180,E1 -6015.638,E2 -6015.638} C_VEL
LIN {X 0,Y 495.682,Z 323.758,A -85,B 0,C 180,E1 -6017.421,E2 -6017.421} C_VEL
LIN {X 0,Y 496.419,Z 329.178,A -85,B 0,C 180,E1 -6017.555,E2 -6017.555} C_VEL
LIN {X 0,Y 497.251,Z 336.663,A -85,B 0,C 180,E1 -6017.685,E2 -6017.685} C_VEL
LIN {X 0,Y 497,Z 399.486,A -85,B 0,C 180,E1 -6018.608,E2 -6018.608} C_VEL
LIN {X 0,Y 496.843,Z 408.633,A -85,B 0,C 180,E1 -6018.837,E2 -6018.837} C_VEL
LIN {X 0,Y 496.639,Z 418.255,A -85,B 0,C 180,E1 -6019.193,E2 -6019.193} C_VEL
LIN {X 0,Y 496.453,Z 428.32,A -85,B 0,C 180,E1 -6019.705,E2 -6019.705} C_VEL
LIN {X 0,Y 496.125,Z 438.767,A -85,B 0,C 180,E1 -6020.419,E2 -6020.419} C_VEL
LIN {X 0,Y 495.836,Z 446.93,A -85,B 0,C 180,E1 -6021.133,E2 -6021.133} C_VEL
LIN {X 0,Y 495.645,Z 453.666,A -85,B 0,C 180,E1 -6021.848,E2 -6021.848} C_VEL
LIN {X 0,Y 495.47,Z 460.044,A -85,B 0,C 180,E1 -6022.666,E2 -6022.666} C_VEL
LIN {X 0,Y 495.371,Z 465.347,A -85,B 0,C 180,E1 -6023.483,E2 -6023.483} C_VEL
LIN {X 0,Y 495.252,Z 469.775,A -85,B 0,C 180,E1 -6024.299,E2 -6024.299} C_VEL
LIN {X 0,Y 495.079,Z 473.465,A -85,B 0,C 180,E1 -6025.114,E2 -6025.114} C_VEL
LIN {X 0,Y 495.104,Z 476.476,A -85,B 0,C 180,E1 -6025.93,E2 -6025.93} C_VEL
LIN {X 0,Y 495.06,Z 478.81,A -85,B 0,C 180,E1 -6026.745,E2 -6026.745} C_VEL
LIN {X 0,Y 495.001,Z 480.589,A -85,B 0,C 180,E1 -6027.559,E2 -6027.559} C_VEL
LIN {X 0,Y 494.961,Z 481.874,A -85,B 0,C 180,E1 -6028.373,E2 -6028.373} C_VEL
LIN {X 0,Y 494.908,Z 482.687,A -85,B 0,C 180,E1 -6029.186,E2 -6029.186} C_VEL
LIN {X 0,Y 494.896,Z 482.997,A -85,B 0,C 180,E1 -6030,E2 -6030} C_VEL
LIN {X 0,Y 494.908,Z 482.723,A -85,B 0,C 180,E1 -6030.814,E2 -6030.814} C_VEL
LIN {X 0,Y 494.961,Z 481.981,A -85,B 0,C 180,E1 -6031.627,E2 -6031.627} C_VEL
LIN {X 0,Y 494.978,Z 480.769,A -85,B 0,C 180,E1 -6032.441,E2 -6032.441} C_VEL
LIN {X 0,Y 495.096,Z 477.914,A -85,B 0,C 180,E1 -6033.662,E2 -6033.662} C_VEL
LIN {X 0,Y 495.085,Z 475.317,A -85,B 0,C 180,E1 -6034.478,E2 -6034.478} C_VEL
LIN {X 0,Y 495.25,Z 470.2,A -85,B 0,C 180,E1 -6035.701,E2 -6035.701} C_VEL
LIN {X 0,Y 495.345,Z 464.814,A -85,B 0,C 180,E1 -6036.701,E2 -6036.701} C_VEL
LIN {X 0,Y 495.515,Z 457.789,A -85,B 0,C 180,E1 -6037.743,E2 -6037.743} C_VEL
LIN {X 0,Y 495.782,Z 449.86,A -85,B 0,C 180,E1 -6038.662,E2 -6038.662} C_VEL
LIN {X 0,Y 496.009,Z 442.299,A -85,B 0,C 180,E1 -6039.378,E2 -6039.378} C_VEL
LIN {X 0,Y 496.211,Z 434.38,A -85,B 0,C 180,E1 -6039.991,E2 -6039.991} C_VEL
LIN {X 0,Y 496.483,Z 426.209,A -85,B 0,C 180,E1 -6040.501,E2 -6040.501} C_VEL
LIN {X 0,Y 496.673,Z 417.943,A -85,B 0,C 180,E1 -6040.909,E2 -6040.909} C_VEL
LIN {X 0,Y 496.831,Z 409.036,A -85,B 0,C 180,E1 -6041.241,E2 -6041.241} C_VEL
LIN {X 0,Y 496.994,Z 400.44,A -85,B 0,C 180,E1 -6041.463,E2 -6041.463} C_VEL
LIN {X 0,Y 497.12,Z 349.292,A -85,B 0,C 180,E1 -6042.226,E2 -6042.226} C_VEL
LIN {X 0,Y 497.057,Z 333.999,A -85,B 0,C 180,E1 -6042.449,E2 -6042.449} C_VEL
LIN {X 0,Y 495.656,Z 323.893,A -85,B 0,C 180,E1 -6042.659,E2 -6042.659} C_VEL
LIN {X 0,Y 495.729,Z 317.532,A -85,B 0,C 180,E1 -6043.946,E2 -6043.946} C_VEL
LIN {X 0,Y 496.098,Z 303.865,A -85,B 0,C 180,E1 -6046.882,E2 -6046.882} C_VEL
LIN {X 0,Y 496.444,Z 292.151,A -85,B 0,C 180,E1 -6049.431,E2 -6049.431} C_VEL
LIN {X 0,Y 496.212,Z 285.975,A -85,B 0,C 180,E1 -6050.807,E2 -6050.807} C_VEL
LIN {X 0,Y 495.797,Z 283.63,A -85,B 0,C 180,E1 -6051.407,E2 -6051.407} C_VEL
LIN {X 0,Y 495.711,Z 283.548,A -85,B 0,C 180,E1 -6054.277,E2 -6054.277} C_VEL
LIN {X 0,Y 495.729,Z 283.544,A -85,B 0,C 180,E1 -6056.979,E2 -6056.979} C_VEL
LIN {X 0,Y 495.756,Z 283.54,A -85,B 0,C 180,E1 -6060.145,E2 -6060.145} C_VEL
LIN {X 0,Y 495.748,Z 283.546,A -85,B 0,C 180,E1 -6063.236,E2 -6063.236} C_VEL
LIN {X 0,Y 495.707,Z 283.546,A -85,B 0,C 180,E1 -6066.086,E2 -6066.086} C_VEL
LIN {X 0,Y 495.754,Z 283.541,A -85,B 0,C 180,E1 -6068.767,E2 -6068.767} C_VEL
LIN {X 0,Y 495.718,Z 283.546,A -85,B 0,C 180,E1 -6071.784,E2 -6071.784} C_VEL
LIN {X 0,Y 495.731,Z 283.551,A -85,B 0,C 180,E1 -6075.14,E2 -6075.14} C_VEL
LIN {X 0,Y 495.717,Z 283.544,A -85,B 0,C 180,E1 -6078.215,E2 -6078.215} C_VEL
LIN {X 0,Y 495.738,Z 283.544,A -85,B 0,C 180,E1 -6081.407,E2 -6081.407} C_VEL
LIN {X 0,Y 495.734,Z 283.545,A -85,B 0,C 180,E1 -6084.461,E2 -6084.461} C_VEL
LIN {X 0,Y 495.742,Z 283.543,A -85,B 0,C 180,E1 -6087.404,E2 -6087.404} C_VEL
LIN {X 0,Y 495.747,Z 283.542,A -85,B 0,C 180,E1 -6090.252,E2 -6090.252} C_VEL
LIN {X 0,Y 495.73,Z 283.544,A -85,B 0,C 180,E1 -6093.27,E2 -6093.27} C_VEL
LIN {X 0,Y 495.727,Z 283.552,A -85,B 0,C 180,E1 -6096.612,E2 -6096.612} C_VEL
LIN {X 0,Y 495.769,Z 283.538,A -85,B 0,C 180,E1 -6099.324,E2 -6099.324} C_VEL
LIN {X 0,Y 495.75,Z 283.541,A -85,B 0,C 180,E1 -6101.827,E2 -6101.827} C_VEL
LIN {X 0,Y 495.765,Z 283.538,A -85,B 0,C 180,E1 -6105.216,E2 -6105.216} C_VEL
LIN {X 0,Y 495.839,Z 283.534,A -85,B 0,C 180,E1 -6108.554,E2 -6108.554} C_VEL
LIN {X 0,Y 495.818,Z 283.535,A -85,B 0,C 180,E1 -6111.851,E2 -6111.851} C_VEL
LIN {X 0,Y 495.843,Z 283.535,A -85,B 0,C 180,E1 -6114.306,E2 -6114.306} C_VEL
LIN {X 0,Y 495.964,Z 283.515,A -85,B 0,C 180,E1 -6117.563,E2 -6117.563} C_VEL
LIN {X 0,Y 495.96,Z 283.522,A -85,B 0,C 180,E1 -6120,E2 -6120} C_VEL
LIN {X 0,Y 495.963,Z 283.516,A -85,B 0,C 180,E1 -6122.436,E2 -6122.436} C_VEL
LIN {X 0,Y 495.842,Z 283.534,A -85,B 0,C 180,E1 -6125.694,E2 -6125.694} C_VEL
LIN {X 0,Y 495.798,Z 283.538,A -85,B 0,C 180,E1 -6128.149,E2 -6128.149} C_VEL
LIN {X 0,Y 495.81,Z 283.537,A -85,B 0,C 180,E1 -6131.446,E2 -6131.446} C_VEL
LIN {X 0,Y 495.764,Z 283.538,A -85,B 0,C 180,E1 -6134.784,E2 -6134.784} C_VEL
LIN {X 0,Y 495.761,Z 283.539,A -85,B 0,C 180,E1 -6138.235,E2 -6138.235} C_VEL
LIN {X 0,Y 495.753,Z 283.54,A -85,B 0,C 180,E1 -6140.757,E2 -6140.757} C_VEL
LIN {X 0,Y 495.723,Z 283.551,A -85,B 0,C 180,E1 -6143.388,E2 -6143.388} C_VEL
LIN {X 0,Y 495.706,Z 283.546,A -85,B 0,C 180,E1 -6146.073,E2 -6146.073} C_VEL
LIN {X 0,Y 495.715,Z 283.547,A -85,B 0,C 180,E1 -6148.818,E2 -6148.818} C_VEL
LIN {X 0,Y 495.74,Z 283.543,A -85,B 0,C 180,E1 -6151.724,E2 -6151.724} C_VEL
LIN {X 0,Y 495.748,Z 283.543,A -85,B 0,C 180,E1 -6154.692,E2 -6154.692} C_VEL
LIN {X 0,Y 495.71,Z 283.547,A -85,B 0,C 180,E1 -6157.563,E2 -6157.563} C_VEL
LIN {X 0,Y 495.735,Z 283.542,A -85,B 0,C 180,E1 -6160.045,E2 -6160.045} C_VEL
LIN {X 0,Y 495.687,Z 283.556,A -85,B 0,C 180,E1 -6162.887,E2 -6162.887} C_VEL
LIN {X 0,Y 495.715,Z 283.544,A -85,B 0,C 180,E1 -6165.998,E2 -6165.998} C_VEL
LIN {X 0,Y 495.72,Z 283.546,A -85,B 0,C 180,E1 -6169.297,E2 -6169.297} C_VEL
LIN {X 0,Y 495.721,Z 283.544,A -85,B 0,C 180,E1 -6171.407,E2 -6171.407} C_VEL
LIN {X 0,Y 495.734,Z 283.548,A -85,B 0,C 180,E1 -6174.462,E2 -6174.462} C_VEL
LIN {X 0,Y 495.746,Z 283.541,A -85,B 0,C 180,E1 -6177.405,E2 -6177.405} C_VEL
LIN {X 0,Y 495.752,Z 283.544,A -85,B 0,C 180,E1 -6180.254,E2 -6180.254} C_VEL
LIN {X 0,Y 495.735,Z 283.542,A -85,B 0,C 180,E1 -6183.271,E2 -6183.271} C_VEL
LIN {X 0,Y 495.735,Z 283.533,A -85,B 0,C 180,E1 -6186.613,E2 -6186.613} C_VEL
LIN {X 0,Y 495.834,Z 283.719,A -85,B 0,C 180,E1 -6188.703,E2 -6188.703} C_VEL
LIN {X 0,Y 496.425,Z 288.045,A -85,B 0,C 180,E1 -6189.706,E2 -6189.706} C_VEL
LIN {X 0,Y 496.297,Z 297.804,A -85,B 0,C 180,E1 -6191.848,E2 -6191.848} C_VEL
LIN {X 0,Y 495.842,Z 313.419,A -85,B 0,C 180,E1 -6195.219,E2 -6195.219} C_VEL
LIN {X 0,Y 495.681,Z 323.781,A -85,B 0,C 180,E1 -6197.378,E2 -6197.378} C_VEL
LIN {X 0,Y 496.635,Z 330.614,A -85,B 0,C 180,E1 -6197.536,E2 -6197.536} C_VEL
LIN {X 0,Y 497.266,Z 337.112,A -85,B 0,C 180,E1 -6197.647,E2 -6197.647} C_VEL
LIN {X 0,Y 496.969,Z 399.369,A -85,B 0,C 180,E1 -6198.56,E2 -6198.56} C_VEL
LIN {X 0,Y 496.82,Z 408.419,A -85,B 0,C 180,E1 -6198.784,E2 -6198.784} C_VEL
LIN {X 0,Y 496.7,Z 416.889,A -85,B 0,C 180,E1 -6199.091,E2 -6199.091} C_VEL
LIN {X 0,Y 496.456,Z 425.392,A -85,B 0,C 180,E1 -6199.499,E2 -6199.499} C_VEL
LIN {X 0,Y 496.245,Z 433.724,A -85,B 0,C 180,E1 -6200.01,E2 -6200.01} C_VEL
LIN {X 0,Y 496.017,Z 441.761,A -85,B 0,C 180,E1 -6200.623,E2 -6200.623} C_VEL
LIN {X 0,Y 495.732,Z 450.433,A -85,B 0,C 180,E1 -6201.439,E2 -6201.439} C_VEL
LIN {X 0,Y 495.48,Z 458.939,A -85,B 0,C 180,E1 -6202.461,E2 -6202.461} C_VEL
LIN {X 0,Y 495.354,Z 465.61,A -85,B 0,C 180,E1 -6203.483,E2 -6203.483} C_VEL
LIN {X 0,Y 495.256,Z 469.989,A -85,B 0,C 180,E1 -6204.299,E2 -6204.299} C_VEL
LIN {X 0,Y 495.086,Z 475.15,A -85,B 0,C 180,E1 -6205.522,E2 -6205.522} C_VEL
LIN {X 0,Y 495.096,Z 477.787,A -85,B 0,C 180,E1 -6206.338,E2 -6206.338} C_VEL
LIN {X 0,Y 495,Z 480.68,A -85,B 0,C 180,E1 -6207.559,E2 -6207.559} C_VEL
LIN {X 0,Y 494.961,Z 481.928,A -85,B 0,C 180,E1 -6208.373,E2 -6208.373} C_VEL
LIN {X 0,Y 494.907,Z 482.706,A -85,B 0,C 180,E1 -6209.186,E2 -6209.186} C_VEL
LIN {X 0,Y 494.895,Z 483,A -85,B 0,C 180,E1 -6210,E2 -6210} C_VEL
LIN {X 0,Y 494.907,Z 482.705,A -85,B 0,C 180,E1 -6210.814,E2 -6210.814} C_VEL
LIN {X 0,Y 494.961,Z 481.927,A -85,B 0,C 180,E1 -6211.627,E2 -6211.627} C_VEL
LIN {X 0,Y 495,Z 480.679,A -85,B 0,C 180,E1 -6212.441,E2 -6212.441} C_VEL
LIN {X 0,Y 495.096,Z 477.786,A -85,B 0,C 180,E1 -6213.662,E2 -6213.662} C_VEL
LIN {X 0,Y 495.086,Z 475.149,A -85,B 0,C 180,E1 -6214.478,E2 -6214.478} C_VEL
LIN {X 0,Y 495.256,Z 469.986,A -85,B 0,C 180,E1 -6215.701,E2 -6215.701} C_VEL
LIN {X 0,Y 495.379,Z 463.45,A -85,B 0,C 180,E1 -6216.885,E2 -6216.885} C_VEL
LIN {X 0,Y 495.577,Z 455.74,A -85,B 0,C 180,E1 -6217.948,E2 -6217.948} C_VEL
LIN {X 0,Y 495.815,Z 448.398,A -85,B 0,C 180,E1 -6218.765,E2 -6218.765} C_VEL
LIN {X 0,Y 496.046,Z 440.535,A -85,B 0,C 180,E1 -6219.48,E2 -6219.48} C_VEL
LIN {X 0,Y 496.292,Z 432.224,A -85,B 0,C 180,E1 -6220.093,E2 -6220.093} C_VEL
LIN {X 0,Y 496.608,Z 421.614,A -85,B 0,C 180,E1 -6220.704,E2 -6220.704} C_VEL
LIN {X 0,Y 496.772,Z 410.082,A -85,B 0,C 180,E1 -6221.165,E2 -6221.165} C_VEL
LIN {X 0,Y 496.934,Z 400.449,A -85,B 0,C 180,E1 -6221.42,E2 -6221.42} C_VEL
LIN {X 0,Y 497.24,Z 336.171,A -85,B 0,C 180,E1 -6222.368,E2 -6222.368} C_VEL
LIN {X 0,Y 495.701,Z 324.065,A -85,B 0,C 180,E1 -6222.601,E2 -6222.601} C_VEL
LIN {X 0,Y 495.662,Z 322.2,A -85,B 0,C 180,E1 -6222.904,E2 -6222.904} C_VEL
LIN {X 0,Y 495.994,Z 307.561,A -85,B 0,C 180,E1 -6226.039,E2 -6226.039} C_VEL
LIN {X 0,Y 496.401,Z 293.896,A -85,B 0,C 180,E1 -6229.003,E2 -6229.003} C_VEL
LIN {X 0,Y 496.42,Z 288.039,A -85,B 0,C 180,E1 -6230.295,E2 -6230.295} C_VEL
LIN {X 0,Y 495.795,Z 283.64,A -85,B 0,C 180,E1 -6231.353,E2 -6231.353} C_VEL
LIN {X 0,Y 495.709,Z 283.548,A -85,B 0,C 180,E1 -6234.277,E2 -6234.277} C_VEL
LIN {X 0,Y 495.727,Z 283.544,A -85,B 0,C 180,E1 -6236.979,E2 -6236.979} C_VEL
LIN {X 0,Y 495.753,Z 283.541,A -85,B 0,C 180,E1 -6240.145,E2 -6240.145} C_VEL
LIN {X 0,Y 495.746,Z 283.546,A -85,B 0,C 180,E1 -6243.236,E2 -6243.236} C_VEL
LIN {X 0,Y 495.702,Z 283.546,A -85,B 0,C 180,E1 -6246.086,E2 -6246.086} C_VEL
LIN {X 0,Y 495.752,Z 283.542,A -85,B 0,C 180,E1 -6248.767,E2 -6248.767} C_VEL
LIN {X 0,Y 495.717,Z 283.546,A -85,B 0,C 180,E1 -6251.784,E2 -6251.784} C_VEL
LIN {X 0,Y 495.73,Z 283.551,A -85,B 0,C 180,E1 -6255.14,E2 -6255.14} C_VEL
LIN {X 0,Y 495.716,Z 283.544,A -85,B 0,C 180,E1 -6258.215,E2 -6258.215} C_VEL
LIN {X 0,Y 495.737,Z 283.544,A -85,B 0,C 180,E1 -6261.407,E2 -6261.407} C_VEL
LIN {X 0,Y 495.73,Z 283.545,A -85,B 0,C 180,E1 -6264.461,E2 -6264.461} C_VEL
LIN {X 0,Y 495.741,Z 283.543,A -85,B 0,C 180,E1 -6267.404,E2 -6267.404} C_VEL
LIN {X 0,Y 495.746,Z 283.543,A -85,B 0,C 180,E1 -6270.252,E2 -6270.252} C_VEL
LIN {X 0,Y 495.729,Z 283.544,A -85,B 0,C 180,E1 -6273.27,E2 -6273.27} C_VEL
LIN {X 0,Y 495.726,Z 283.551,A -85,B 0,C 180,E1 -6276.612,E2 -6276.612} C_VEL
LIN {X 0,Y 495.768,Z 283.538,A -85,B 0,C 180,E1 -6279.324,E2 -6279.324} C_VEL
LIN {X 0,Y 495.75,Z 283.541,A -85,B 0,C 180,E1 -6281.827,E2 -6281.827} C_VEL
LIN {X 0,Y 495.764,Z 283.538,A -85,B 0,C 180,E1 -6285.216,E2 -6285.216} C_VEL
LIN {X 0,Y 495.839,Z 283.534,A -85,B 0,C 180,E1 -6288.555,E2 -6288.555} C_VEL
LIN {X 0,Y 495.801,Z 283.537,A -85,B 0,C 180,E1 -6291.851,E2 -6291.851} C_VEL
LIN {X 0,Y 495.843,Z 283.535,A -85,B 0,C 180,E1 -6294.306,E2 -6294.306} C_VEL
LIN {X 0,Y 495.964,Z 283.515,A -85,B 0,C 180,E1 -6297.564,E2 -6297.564} C_VEL
LIN {X 0,Y 495.96,Z 283.522,A -85,B 0,C 180,E1 -6300,E2 -6300} C_VEL
LIN {X 0,Y 495.963,Z 283.516,A -85,B 0,C 180,E1 -6302.437,E2 -6302.437} C_VEL
LIN {X 0,Y 495.843,Z 283.534,A -85,B 0,C 180,E1 -6305.694,E2 -6305.694} C_VEL
LIN {X 0,Y 495.798,Z 283.538,A -85,B 0,C 180,E1 -6308.149,E2 -6308.149} C_VEL
LIN {X 0,Y 495.81,Z 283.537,A -85,B 0,C 180,E1 -6311.446,E2 -6311.446} C_VEL
LIN {X 0,Y 495.763,Z 283.538,A -85,B 0,C 180,E1 -6314.784,E2 -6314.784} C_VEL
LIN {X 0,Y 495.762,Z 283.539,A -85,B 0,C 180,E1 -6318.235,E2 -6318.235} C_VEL
LIN {X 0,Y 495.754,Z 283.54,A -85,B 0,C 180,E1 -6320.757,E2 -6320.757} C_VEL
LIN {X 0,Y 495.724,Z 283.551,A -85,B 0,C 180,E1 -6323.389,E2 -6323.389} C_VEL
LIN {X 0,Y 495.706,Z 283.546,A -85,B 0,C 180,E1 -6326.073,E2 -6326.073} C_VEL
LIN {X 0,Y 495.708,Z 283.547,A -85,B 0,C 180,E1 -6328.819,E2 -6328.819} C_VEL
LIN {X 0,Y 495.729,Z 283.545,A -85,B 0,C 180,E1 -6331.722,E2 -6331.722} C_VEL
LIN {X 0,Y 495.748,Z 283.542,A -85,B 0,C 180,E1 -6334.692,E2 -6334.692} C_VEL
LIN {X 0,Y 495.704,Z 283.548,A -85,B 0,C 180,E1 -6337.564,E2 -6337.564} C_VEL
LIN {X 0,Y 495.736,Z 283.542,A -85,B 0,C 180,E1 -6340.045,E2 -6340.045} C_VEL
LIN {X 0,Y 495.688,Z 283.555,A -85,B 0,C 180,E1 -6342.887,E2 -6342.887} C_VEL
LIN {X 0,Y 495.716,Z 283.544,A -85,B 0,C 180,E1 -6345.998,E2 -6345.998} C_VEL
LIN {X 0,Y 495.72,Z 283.546,A -85,B 0,C 180,E1 -6349.297,E2 -6349.297} C_VEL
LIN {X 0,Y 495.722,Z 283.545,A -85,B 0,C 180,E1 -6351.407,E2 -6351.407} C_VEL
LIN {X 0,Y 495.735,Z 283.547,A -85,B 0,C 180,E1 -6354.462,E2 -6354.462} C_VEL
LIN {X 0,Y 495.747,Z 283.541,A -85,B 0,C 180,E1 -6357.405,E2 -6357.405} C_VEL
LIN {X 0,Y 495.707,Z 283.55,A -85,B 0,C 180,E1 -6360.251,E2 -6360.251} C_VEL
LIN {X 0,Y 495.684,Z 283.549,A -85,B 0,C 180,E1 -6360.715,E2 -6360.715} C_VEL
LIN {X 0,Y 495.014,Z 283.634,A -85,B 0,C 180,E1 -6361.394,E2 -6361.394} C_VEL
LIN {X 0,Y 492.155,Z 283.997,A -85,B 0,C 180,E1 -6362.496,E2 -6362.496} C_VEL
LIN {X 0,Y 489.755,Z 284.291,A -85,B 0,C 180,E1 -6363.385,E2 -6363.385} C_VEL
LIN {X 0,Y 488.748,Z 284.416,A -85,B 0,C 180,E1 -6364.071,E2 -6364.071} C_VEL
LIN {X 0,Y 488.679,Z 284.427,A -85,B 0,C 180,E1 -6364.304,E2 -6364.304} C_VEL
LIN {X 0,Y 488.705,Z 284.404,A -85,B 0,C 180,E1 -6367.153,E2 -6367.153} C_VEL
LIN {X 0,Y 488.791,Z 284.69,A -85,B 0,C 180,E1 -6368.657,E2 -6368.657} C_VEL
LIN {X 0,Y 489.434,Z 289.792,A -85,B 0,C 180,E1 -6369.842,E2 -6369.842} C_VEL
LIN {X 0,Y 489.251,Z 299.55,A -85,B 0,C 180,E1 -6372.011,E2 -6372.011} C_VEL
LIN {X 0,Y 488.78,Z 315.162,A -85,B 0,C 180,E1 -6375.427,E2 -6375.427} C_VEL
LIN {X 0,Y 488.639,Z 323.703,A -85,B 0,C 180,E1 -6377.228,E2 -6377.228} C_VEL
LIN {X 0,Y 489.17,Z 327.777,A -85,B 0,C 180,E1 -6377.347,E2 -6377.347} C_VEL
LIN {X 0,Y 490.331,Z 336.005,A -85,B 0,C 180,E1 -6377.498,E2 -6377.498} C_VEL
LIN {X 0,Y 490.066,Z 399.512,A -85,B 0,C 180,E1 -6378.444,E2 -6378.444} C_VEL
LIN {X 0,Y 489.892,Z 408.65,A -85,B 0,C 180,E1 -6378.676,E2 -6378.676} C_VEL
LIN {X 0,Y 489.686,Z 418.267,A -85,B 0,C 180,E1 -6379.038,E2 -6379.038} C_VEL
LIN {X 0,Y 489.448,Z 428.329,A -85,B 0,C 180,E1 -6379.556,E2 -6379.556} C_VEL
LIN {X 0,Y 489.128,Z 438.773,A -85,B 0,C 180,E1 -6380.28,E2 -6380.28} C_VEL
LIN {X 0,Y 488.826,Z 446.936,A -85,B 0,C 180,E1 -6381.005,E2 -6381.005} C_VEL
LIN {X 0,Y 488.607,Z 453.671,A -85,B 0,C 180,E1 -6381.73,E2 -6381.73} C_VEL
LIN {X 0,Y 488.423,Z 460.048,A -85,B 0,C 180,E1 -6382.559,E2 -6382.559} C_VEL
LIN {X 0,Y 488.307,Z 466.143,A -85,B 0,C 180,E1 -6383.529,E2 -6383.529} C_VEL
LIN {X 0,Y 488.189,Z 469.778,A -85,B 0,C 180,E1 -6384.216,E2 -6384.216} C_VEL
LIN {X 0,Y 487.993,Z 474.984,A -85,B 0,C 180,E1 -6385.457,E2 -6385.457} C_VEL
LIN {X 0,Y 488.023,Z 477.661,A -85,B 0,C 180,E1 -6386.284,E2 -6386.284} C_VEL
LIN {X 0,Y 487.912,Z 480.591,A -85,B 0,C 180,E1 -6387.523,E2 -6387.523} C_VEL
LIN {X 0,Y 487.89,Z 481.875,A -85,B 0,C 180,E1 -6388.349,E2 -6388.349} C_VEL
LIN {X 0,Y 487.831,Z 482.688,A -85,B 0,C 180,E1 -6389.175,E2 -6389.175} C_VEL
LIN {X 0,Y 487.817,Z 482.997,A -85,B 0,C 180,E1 -6390,E2 -6390} C_VEL
LIN {X 0,Y 487.832,Z 482.723,A -85,B 0,C 180,E1 -6390.825,E2 -6390.825} C_VEL
LIN {X 0,Y 487.888,Z 481.981,A -85,B 0,C 180,E1 -6391.651,E2 -6391.651} C_VEL
LIN {X 0,Y 487.891,Z 480.768,A -85,B 0,C 180,E1 -6392.477,E2 -6392.477} C_VEL
LIN {X 0,Y 488.021,Z 477.912,A -85,B 0,C 180,E1 -6393.716,E2 -6393.716} C_VEL
LIN {X 0,Y 487.988,Z 475.315,A -85,B 0,C 180,E1 -6394.543,E2 -6394.543} C_VEL
LIN {X 0,Y 488.179,Z 470.197,A -85,B 0,C 180,E1 -6395.784,E2 -6395.784} C_VEL
LIN {X 0,Y 488.273,Z 465.338,A -85,B 0,C 180,E1 -6396.705,E2 -6396.705} C_VEL
LIN {X 0,Y 488.477,Z 457.785,A -85,B 0,C 180,E1 -6397.856,E2 -6397.856} C_VEL
LIN {X 0,Y 488.748,Z 449.854,A -85,B 0,C 180,E1 -6398.788,E2 -6398.788} C_VEL
LIN {X 0,Y 488.985,Z 442.292,A -85,B 0,C 180,E1 -6399.514,E2 -6399.514} C_VEL
LIN {X 0,Y 489.23,Z 434.372,A -85,B 0,C 180,E1 -6400.135,E2 -6400.135} C_VEL
LIN {X 0,Y 489.499,Z 426.199,A -85,B 0,C 180,E1 -6400.652,E2 -6400.652} C_VEL
LIN {X 0,Y 489.688,Z 417.931,A -85,B 0,C 180,E1 -6401.067,E2 -6401.067} C_VEL
LIN {X 0,Y 489.873,Z 409.02,A -85,B 0,C 180,E1 -6401.403,E2 -6401.403} C_VEL
LIN {X 0,Y 490.039,Z 399.439,A -85,B 0,C 180,E1 -6401.648,E2 -6401.648} C_VEL
LIN {X 0,Y 490.209,Z 335.106,A -85,B 0,C 180,E1 -6402.609,E2 -6402.609} C_VEL
LIN {X 0,Y 488.627,Z 323.887,A -85,B 0,C 180,E1 -6402.844,E2 -6402.844} C_VEL
LIN {X 0,Y 488.707,Z 317.53,A -85,B 0,C 180,E1 -6404.15,E2 -6404.15} C_VEL
LIN {X 0,Y 489.103,Z 303.863,A -85,B 0,C 180,E1 -6407.131,E2 -6407.131} C_VEL
LIN {X 0,Y 489.472,Z 292.149,A -85,B 0,C 180,E1 -6409.719,E2 -6409.719} C_VEL
LIN {X 0,Y 489.078,Z 286.291,A -85,B 0,C 180,E1 -6411.053,E2 -6411.053} C_VEL
LIN {X 0,Y 488.77,Z 284.518,A -85,B 0,C 180,E1 -6411.509,E2 -6411.509} C_VEL
LIN {X 0,Y 488.695,Z 284.421,A -85,B 0,C 180,E1 -6414.648,E2 -6414.648} C_VEL
LIN {X 0,Y 488.682,Z 284.426,A -85,B 0,C 180,E1 -6417.4,E2 -6417.4} C_VEL
LIN {X 0,Y 488.701,Z 284.418,A -85,B 0,C 180,E1 -6420.361,E2 -6420.361} C_VEL
LIN {X 0,Y 488.707,Z 284.425,A -85,B 0,C 180,E1 -6423.479,E2 -6423.479} C_VEL
LIN {X 0,Y 488.669,Z 284.422,A -85,B 0,C 180,E1 -6426.352,E2 -6426.352} C_VEL
LIN {X 0,Y 488.69,Z 284.428,A -85,B 0,C 180,E1 -6429.254,E2 -6429.254} C_VEL
LIN {X 0,Y 488.644,Z 284.426,A -85,B 0,C 180,E1 -6432.529,E2 -6432.529} C_VEL
LIN {X 0,Y 488.695,Z 284.427,A -85,B 0,C 180,E1 -6435.196,E2 -6435.196} C_VEL
LIN {X 0,Y 488.655,Z 284.426,A -85,B 0,C 180,E1 -6438.579,E2 -6438.579} C_VEL
LIN {X 0,Y 488.691,Z 284.427,A -85,B 0,C 180,E1 -6440.948,E2 -6440.948} C_VEL
LIN {X 0,Y 488.661,Z 284.423,A -85,B 0,C 180,E1 -6443.866,E2 -6443.866} C_VEL
LIN {X 0,Y 488.693,Z 284.427,A -85,B 0,C 180,E1 -6446.874,E2 -6446.874} C_VEL
LIN {X 0,Y 488.707,Z 284.417,A -85,B 0,C 180,E1 -6449.779,E2 -6449.779} C_VEL
LIN {X 0,Y 488.688,Z 284.423,A -85,B 0,C 180,E1 -6453.078,E2 -6453.078} C_VEL
LIN {X 0,Y 488.657,Z 284.427,A -85,B 0,C 180,E1 -6456.253,E2 -6456.253} C_VEL
LIN {X 0,Y 488.711,Z 284.418,A -85,B 0,C 180,E1 -6459.183,E2 -6459.183} C_VEL
LIN {X 0,Y 488.737,Z 284.414,A -85,B 0,C 180,E1 -6461.632,E2 -6461.632} C_VEL
LIN {X 0,Y 488.736,Z 284.415,A -85,B 0,C 180,E1 -6464.999,E2 -6464.999} C_VEL
LIN {X 0,Y 488.794,Z 284.414,A -85,B 0,C 180,E1 -6468.387,E2 -6468.387} C_VEL
LIN {X 0,Y 488.767,Z 284.412,A -85,B 0,C 180,E1 -6471.733,E2 -6471.733} C_VEL
LIN {X 0,Y 488.803,Z 284.413,A -85,B 0,C 180,E1 -6474.224,E2 -6474.224} C_VEL
LIN {X 0,Y 488.93,Z 284.391,A -85,B 0,C 180,E1 -6477.528,E2 -6477.528} C_VEL
LIN {X 0,Y 488.929,Z 284.398,A -85,B 0,C 180,E1 -6480,E2 -6480} C_VEL
LIN {X 0,Y 488.929,Z 284.392,A -85,B 0,C 180,E1 -6482.471,E2 -6482.471} C_VEL
LIN {X 0,Y 488.802,Z 284.413,A -85,B 0,C 180,E1 -6485.776,E2 -6485.776} C_VEL
LIN {X 0,Y 488.744,Z 284.415,A -85,B 0,C 180,E1 -6488.268,E2 -6488.268} C_VEL
LIN {X 0,Y 488.772,Z 284.416,A -85,B 0,C 180,E1 -6491.613,E2 -6491.613} C_VEL
LIN {X 0,Y 488.735,Z 284.415,A -85,B 0,C 180,E1 -6495.001,E2 -6495.001} C_VEL
LIN {X 0,Y 488.733,Z 284.414,A -85,B 0,C 180,E1 -6498.443,E2 -6498.443} C_VEL
LIN {X 0,Y 488.689,Z 284.422,A -85,B 0,C 180,E1 -6501.071,E2 -6501.071} C_VEL
LIN {X 0,Y 488.654,Z 284.428,A -85,B 0,C 180,E1 -6503.747,E2 -6503.747} C_VEL
LIN {X 0,Y 488.671,Z 284.422,A -85,B 0,C 180,E1 -6506.477,E2 -6506.477} C_VEL
LIN {X 0,Y 488.689,Z 284.428,A -85,B 0,C 180,E1 -6509.273,E2 -6509.273} C_VEL
LIN {X 0,Y 488.685,Z 284.42,A -85,B 0,C 180,E1 -6512.148,E2 -6512.148} C_VEL
LIN {X 0,Y 488.701,Z 284.426,A -85,B 0,C 180,E1 -6515.116,E2 -6515.116} C_VEL
LIN {X 0,Y 488.665,Z 284.423,A -85,B 0,C 180,E1 -6518.201,E2 -6518.201} C_VEL
LIN {X 0,Y 488.686,Z 284.421,A -85,B 0,C 180,E1 -6520.342,E2 -6520.342} C_VEL
LIN {X 0,Y 488.665,Z 284.423,A -85,B 0,C 180,E1 -6523.657,E2 -6523.657} C_VEL
LIN {X 0,Y 488.666,Z 284.424,A -85,B 0,C 180,E1 -6526.345,E2 -6526.345} C_VEL
LIN {X 0,Y 488.698,Z 284.419,A -85,B 0,C 180,E1 -6529.674,E2 -6529.674} C_VEL
LIN {X 0,Y 488.659,Z 284.43,A -85,B 0,C 180,E1 -6532.84,E2 -6532.84} C_VEL
LIN {X 0,Y 488.712,Z 284.417,A -85,B 0,C 180,E1 -6535.887,E2 -6535.887} C_VEL
LIN {X 0,Y 488.681,Z 284.425,A -85,B 0,C 180,E1 -6538.82,E2 -6538.82} C_VEL
LIN {X 0,Y 488.689,Z 284.42,A -85,B 0,C 180,E1 -6541.668,E2 -6541.668} C_VEL
LIN {X 0,Y 488.695,Z 284.423,A -85,B 0,C 180,E1 -6544.96,E2 -6544.96} C_VEL
LIN {X 0,Y 488.774,Z 284.49,A -85,B 0,C 180,E1 -6548.491,E2 -6548.491} C_VEL
LIN {X 0,Y 488.885,Z 285.12,A -85,B 0,C 180,E1 -6548.717,E2 -6548.717} C_VEL
LIN {X 0,Y 489.473,Z 289.998,A -85,B 0,C 180,E1 -6549.843,E2 -6549.843} C_VEL
LIN {X 0,Y 489.163,Z 301.708,A -85,B 0,C 180,E1 -6552.44,E2 -6552.44} C_VEL
LIN {X 0,Y 488.778,Z 315.371,A -85,B 0,C 180,E1 -6555.427,E2 -6555.427} C_VEL
LIN {X 0,Y 488.644,Z 323.782,A -85,B 0,C 180,E1 -6557.193,E2 -6557.193} C_VEL
LIN {X 0,Y 489.582,Z 330.144,A -85,B 0,C 180,E1 -6557.347,E2 -6557.347} C_VEL
LIN {X 0,Y 490.35,Z 337.122,A -85,B 0,C 180,E1 -6557.47,E2 -6557.47} C_VEL
LIN {X 0,Y 490.01,Z 399.424,A -85,B 0,C 180,E1 -6558.396,E2 -6558.396} C_VEL
LIN {X 0,Y 489.876,Z 408.423,A -85,B 0,C 180,E1 -6558.623,E2 -6558.623} C_VEL
LIN {X 0,Y 489.743,Z 416.892,A -85,B 0,C 180,E1 -6558.934,E2 -6558.934} C_VEL
LIN {X 0,Y 489.481,Z 425.394,A -85,B 0,C 180,E1 -6559.347,E2 -6559.347} C_VEL
LIN {X 0,Y 489.248,Z 433.726,A -85,B 0,C 180,E1 -6559.865,E2 -6559.865} C_VEL
LIN {X 0,Y 488.993,Z 441.762,A -85,B 0,C 180,E1 -6560.487,E2 -6560.487} C_VEL
LIN {X 0,Y 488.7,Z 450.434,A -85,B 0,C 180,E1 -6561.315,E2 -6561.315} C_VEL
LIN {X 0,Y 488.432,Z 458.939,A -85,B 0,C 180,E1 -6562.352,E2 -6562.352} C_VEL
LIN {X 0,Y 488.288,Z 465.61,A -85,B 0,C 180,E1 -6563.388,E2 -6563.388} C_VEL
LIN {X 0,Y 488.19,Z 469.989,A -85,B 0,C 180,E1 -6564.216,E2 -6564.216} C_VEL
LIN {X 0,Y 487.989,Z 475.15,A -85,B 0,C 180,E1 -6565.457,E2 -6565.457} C_VEL
LIN {X 0,Y 487.986,Z 478.938,A -85,B 0,C 180,E1 -6566.698,E2 -6566.698} C_VEL
LIN {X 0,Y 487.911,Z 480.68,A -85,B 0,C 180,E1 -6567.523,E2 -6567.523} C_VEL
LIN {X 0,Y 487.889,Z 481.928,A -85,B 0,C 180,E1 -6568.349,E2 -6568.349} C_VEL
LIN {X 0,Y 487.831,Z 482.706,A -85,B 0,C 180,E1 -6569.175,E2 -6569.175} C_VEL
LIN {X 0,Y 487.816,Z 483,A -85,B 0,C 180,E1 -6570,E2 -6570} C_VEL
LIN {X 0,Y 487.831,Z 482.705,A -85,B 0,C 180,E1 -6570.825,E2 -6570.825} C_VEL
LIN {X 0,Y 487.889,Z 481.927,A -85,B 0,C 180,E1 -6571.651,E2 -6571.651} C_VEL
LIN {X 0,Y 487.911,Z 480.679,A -85,B 0,C 180,E1 -6572.477,E2 -6572.477} C_VEL
LIN {X 0,Y 488.021,Z 477.786,A -85,B 0,C 180,E1 -6573.716,E2 -6573.716} C_VEL
LIN {X 0,Y 487.989,Z 475.149,A -85,B 0,C 180,E1 -6574.543,E2 -6574.543} C_VEL
LIN {X 0,Y 488.189,Z 469.986,A -85,B 0,C 180,E1 -6575.784,E2 -6575.784} C_VEL
LIN {X 0,Y 488.314,Z 463.45,A -85,B 0,C 180,E1 -6576.985,E2 -6576.985} C_VEL
LIN {X 0,Y 488.537,Z 455.74,A -85,B 0,C 180,E1 -6578.063,E2 -6578.063} C_VEL
LIN {X 0,Y 488.793,Z 448.397,A -85,B 0,C 180,E1 -6578.891,E2 -6578.891} C_VEL
LIN {X 0,Y 489.038,Z 440.533,A -85,B 0,C 180,E1 -6579.617,E2 -6579.617} C_VEL
LIN {X 0,Y 489.316,Z 432.222,A -85,B 0,C 180,E1 -6580.238,E2 -6580.238} C_VEL
LIN {X 0,Y 489.626,Z 421.611,A -85,B 0,C 180,E1 -6580.859,E2 -6580.859} C_VEL
LIN {X 0,Y 489.83,Z 410.078,A -85,B 0,C 180,E1 -6581.325,E2 -6581.325} C_VEL
LIN {X 0,Y 489.998,Z 400.442,A -85,B 0,C 180,E1 -6581.584,E2 -6581.584} C_VEL
LIN {X 0,Y 490.254,Z 335.405,A -85,B 0,C 180,E1 -6582.558,E2 -6582.558} C_VEL
LIN {X 0,Y 488.67,Z 324.063,A -85,B 0,C 180,E1 -6582.785,E2 -6582.785} C_VEL
LIN {X 0,Y 488.606,Z 322.2,A -85,B 0,C 180,E1 -6583.094,E2 -6583.094} C_VEL
LIN {X 0,Y 488.989,Z 307.56,A -85,B 0,C 180,E1 -6586.276,E2 -6586.276} C_VEL
LIN {X 0,Y 489.424,Z 293.895,A -85,B 0,C 180,E1 -6589.285,E2 -6589.285} C_VEL
LIN {X 0,Y 489.366,Z 288.287,A -85,B 0,C 180,E1 -6590.544,E2 -6590.544} C_VEL
LIN {X 0,Y 488.738,Z 284.531,A -85,B 0,C 180,E1 -6591.456,E2 -6591.456} C_VEL
LIN {X 0,Y 488.693,Z 284.421,A -85,B 0,C 180,E1 -6594.648,E2 -6594.648} C_VEL
LIN {X 0,Y 488.68,Z 284.427,A -85,B 0,C 180,E1 -6597.4,E2 -6597.4} C_VEL
LIN {X 0,Y 488.697,Z 284.419,A -85,B 0,C 180,E1 -6600.36,E2 -6600.36} C_VEL
LIN {X 0,Y 488.705,Z 284.425,A -85,B 0,C 180,E1 -6603.479,E2 -6603.479} C_VEL
LIN {X 0,Y 488.664,Z 284.423,A -85,B 0,C 180,E1 -6606.352,E2 -6606.352} C_VEL
LIN {X 0,Y 488.688,Z 284.428,A -85,B 0,C 180,E1 -6609.254,E2 -6609.254} C_VEL
LIN {X 0,Y 488.661,Z 284.426,A -85,B 0,C 180,E1 -6611.594,E2 -6611.594} C_VEL
LIN {X 0,Y 488.694,Z 284.423,A -85,B 0,C 180,E1 -6614.802,E2 -6614.802} C_VEL
LIN {X 0,Y 488.642,Z 284.428,A -85,B 0,C 180,E1 -6617.469,E2 -6617.469} C_VEL
LIN {X 0,Y 488.696,Z 284.42,A -85,B 0,C 180,E1 -6619.673,E2 -6619.673} C_VEL
LIN {X 0,Y 488.659,Z 284.431,A -85,B 0,C 180,E1 -6622.839,E2 -6622.839} C_VEL
LIN {X 0,Y 488.708,Z 284.417,A -85,B 0,C 180,E1 -6625.885,E2 -6625.885} C_VEL
LIN {X 0,Y 488.676,Z 284.429,A -85,B 0,C 180,E1 -6628.819,E2 -6628.819} C_VEL
LIN {X 0,Y 488.683,Z 284.42,A -85,B 0,C 180,E1 -6631.667,E2 -6631.667} C_VEL
LIN {X 0,Y 488.688,Z 284.424,A -85,B 0,C 180,E1 -6634.959,E2 -6634.959} C_VEL
LIN {X 0,Y 488.678,Z 284.423,A -85,B 0,C 180,E1 -6638.042,E2 -6638.042} C_VEL
LIN {X 0,Y 488.715,Z 284.422,A -85,B 0,C 180,E1 -6640.686,E2 -6640.686} C_VEL
LIN {X 0,Y 488.658,Z 284.423,A -85,B 0,C 180,E1 -6643.283,E2 -6643.283} C_VEL
LIN {X 0,Y 488.709,Z 284.419,A -85,B 0,C 180,E1 -6645.849,E2 -6645.849} C_VEL
LIN {X 0,Y 488.793,Z 284.414,A -85,B 0,C 180,E1 -6648.387,E2 -6648.387} C_VEL
LIN {X 0,Y 488.749,Z 284.414,A -85,B 0,C 180,E1 -6651.733,E2 -6651.733} C_VEL
LIN {X 0,Y 488.803,Z 284.413,A -85,B 0,C 180,E1 -6654.224,E2 -6654.224} C_VEL
LIN {X 0,Y 488.93,Z 284.391,A -85,B 0,C 180,E1 -6657.529,E2 -6657.529} C_VEL
LIN {X 0,Y 488.929,Z 284.398,A -85,B 0,C 180,E1 -6660,E2 -6660} C_VEL
LIN {X 0,Y 488.929,Z 284.392,A -85,B 0,C 180,E1 -6662.472,E2 -6662.472} C_VEL
LIN {X 0,Y 488.802,Z 284.412,A -85,B 0,C 180,E1 -6665.776,E2 -6665.776} C_VEL
LIN {X 0,Y 488.742,Z 284.416,A -85,B 0,C 180,E1 -6668.268,E2 -6668.268} C_VEL
LIN {X 0,Y 488.772,Z 284.416,A -85,B 0,C 180,E1 -6671.613,E2 -6671.613} C_VEL
LIN {X 0,Y 488.735,Z 284.415,A -85,B 0,C 180,E1 -6675.001,E2 -6675.001} C_VEL
LIN {X 0,Y 488.733,Z 284.414,A -85,B 0,C 180,E1 -6678.443,E2 -6678.443} C_VEL
LIN {X 0,Y 488.69,Z 284.422,A -85,B 0,C 180,E1 -6681.072,E2 -6681.072} C_VEL
LIN {X 0,Y 488.655,Z 284.428,A -85,B 0,C 180,E1 -6683.748,E2 -6683.748} C_VEL
LIN {X 0,Y 488.671,Z 284.422,A -85,B 0,C 180,E1 -6686.477,E2 -6686.477} C_VEL
LIN {X 0,Y 488.678,Z 284.429,A -85,B 0,C 180,E1 -6689.273,E2 -6689.273} C_VEL
LIN {X 0,Y 488.681,Z 284.421,A -85,B 0,C 180,E1 -6692.149,E2 -6692.149} C_VEL
LIN {X 0,Y 488.702,Z 284.426,A -85,B 0,C 180,E1 -6695.116,E2 -6695.116} C_VEL
LIN {X 0,Y 488.654,Z 284.424,A -85,B 0,C 180,E1 -6698.203,E2 -6698.203} C_VEL
LIN {X 0,Y 488.687,Z 284.421,A -85,B 0,C 180,E1 -6700.342,E2 -6700.342} C_VEL
LIN {X 0,Y 488.666,Z 284.423,A -85,B 0,C 180,E1 -6703.657,E2 -6703.657} C_VEL
LIN {X 0,Y 488.667,Z 284.424,A -85,B 0,C 180,E1 -6706.345,E2 -6706.345} C_VEL
LIN {X 0,Y 488.699,Z 284.418,A -85,B 0,C 180,E1 -6709.674,E2 -6709.674} C_VEL
LIN {X 0,Y 488.661,Z 284.43,A -85,B 0,C 180,E1 -6712.84,E2 -6712.84} C_VEL
LIN {X 0,Y 488.713,Z 284.417,A -85,B 0,C 180,E1 -6715.887,E2 -6715.887} C_VEL
LIN {X 0,Y 488.671,Z 284.427,A -85,B 0,C 180,E1 -6718.82,E2 -6718.82} C_VEL
LIN {X 0,Y 488.683,Z 284.42,A -85,B 0,C 180,E1 -6721.668,E2 -6721.668} C_VEL
LIN {X 0,Y 488.679,Z 284.427,A -85,B 0,C 180,E1 -6724.304,E2 -6724.304} C_VEL
LIN {X 0,Y 488.039,Z 284.511,A -85,B 0,C 180,E1 -6724.991,E2 -6724.991} C_VEL
LIN {X 0,Y 485.171,Z 284.858,A -85,B 0,C 180,E1 -6726.108,E2 -6726.108} C_VEL
LIN {X 0,Y 482.743,Z 285.148,A -85,B 0,C 180,E1 -6727.008,E2 -6727.008} C_VEL
LIN {X 0,Y 481.722,Z 285.27,A -85,B 0,C 180,E1 -6727.704,E2 -6727.704} C_VEL
LIN {X 0,Y 481.651,Z 285.279,A -85,B 0,C 180,E1 -6727.94,E2 -6727.94} C_VEL
LIN {X 0,Y 481.721,Z 285.47,A -85,B 0,C 180,E1 -6728.497,E2 -6728.497} C_VEL
LIN {X 0,Y 482.443,Z 291.746,A -85,B 0,C 180,E1 -6729.981,E2 -6729.981} C_VEL
LIN {X 0,Y 482.181,Z 301.503,A -85,B 0,C 180,E1 -6732.177,E2 -6732.177} C_VEL
LIN {X 0,Y 481.764,Z 315.165,A -85,B 0,C 180,E1 -6735.21,E2 -6735.21} C_VEL
LIN {X 0,Y 481.575,Z 323.642,A -85,B 0,C 180,E1 -6737.029,E2 -6737.029} C_VEL
LIN {X 0,Y 481.936,Z 326.358,A -85,B 0,C 180,E1 -6737.132,E2 -6737.132} C_VEL
LIN {X 0,Y 483.377,Z 336.183,A -85,B 0,C 180,E1 -6737.317,E2 -6737.317} C_VEL
LIN {X 0,Y 483.138,Z 399.535,A -85,B 0,C 180,E1 -6738.276,E2 -6738.276} C_VEL
LIN {X 0,Y 482.939,Z 408.665,A -85,B 0,C 180,E1 -6738.511,E2 -6738.511} C_VEL
LIN {X 0,Y 482.755,Z 417.068,A -85,B 0,C 180,E1 -6738.825,E2 -6738.825} C_VEL
LIN {X 0,Y 482.509,Z 424.594,A -85,B 0,C 180,E1 -6739.192,E2 -6739.192} C_VEL
LIN {X 0,Y 482.313,Z 433.083,A -85,B 0,C 180,E1 -6739.718,E2 -6739.718} C_VEL
LIN {X 0,Y 482.031,Z 441.239,A -85,B 0,C 180,E1 -6740.348,E2 -6740.348} C_VEL
LIN {X 0,Y 481.754,Z 448.982,A -85,B 0,C 180,E1 -6741.083,E2 -6741.083} C_VEL
LIN {X 0,Y 481.44,Z 457.077,A -85,B 0,C 180,E1 -6742.029,E2 -6742.029} C_VEL
LIN {X 0,Y 481.309,Z 463.163,A -85,B 0,C 180,E1 -6742.913,E2 -6742.913} C_VEL
LIN {X 0,Y 481.127,Z 469.78,A -85,B 0,C 180,E1 -6744.131,E2 -6744.131} C_VEL
LIN {X 0,Y 480.904,Z 474.986,A -85,B 0,C 180,E1 -6745.39,E2 -6745.39} C_VEL
LIN {X 0,Y 480.948,Z 477.662,A -85,B 0,C 180,E1 -6746.23,E2 -6746.23} C_VEL
LIN {X 0,Y 480.827,Z 480.592,A -85,B 0,C 180,E1 -6747.487,E2 -6747.487} C_VEL
LIN {X 0,Y 480.791,Z 481.875,A -85,B 0,C 180,E1 -6748.325,E2 -6748.325} C_VEL
LIN {X 0,Y 480.757,Z 482.688,A -85,B 0,C 180,E1 -6749.162,E2 -6749.162} C_VEL
LIN {X 0,Y 480.741,Z 482.997,A -85,B 0,C 180,E1 -6750,E2 -6750} C_VEL
LIN {X 0,Y 480.758,Z 482.723,A -85,B 0,C 180,E1 -6750.838,E2 -6750.838} C_VEL
LIN {X 0,Y 480.789,Z 481.98,A -85,B 0,C 180,E1 -6751.675,E2 -6751.675} C_VEL
LIN {X 0,Y 480.808,Z 480.767,A -85,B 0,C 180,E1 -6752.513,E2 -6752.513} C_VEL
LIN {X 0,Y 480.945,Z 477.911,A -85,B 0,C 180,E1 -6753.77,E2 -6753.77} C_VEL
LIN {X 0,Y 480.899,Z 475.313,A -85,B 0,C 180,E1 -6754.61,E2 -6754.61} C_VEL
LIN {X 0,Y 481.113,Z 470.194,A -85,B 0,C 180,E1 -6755.869,E2 -6755.869} C_VEL
LIN {X 0,Y 481.289,Z 463.476,A -85,B 0,C 180,E1 -6757.13,E2 -6757.13} C_VEL
LIN {X 0,Y 481.479,Z 456.103,A -85,B 0,C 180,E1 -6758.182,E2 -6758.182} C_VEL
LIN {X 0,Y 481.754,Z 448.829,A -85,B 0,C 180,E1 -6759.022,E2 -6759.022} C_VEL
LIN {X 0,Y 482.054,Z 441.057,A -85,B 0,C 180,E1 -6759.758,E2 -6759.758} C_VEL
LIN {X 0,Y 482.303,Z 432.864,A -85,B 0,C 180,E1 -6760.388,E2 -6760.388} C_VEL
LIN {X 0,Y 482.532,Z 424.318,A -85,B 0,C 180,E1 -6760.914,E2 -6760.914} C_VEL
LIN {X 0,Y 482.839,Z 413.029,A -85,B 0,C 180,E1 -6761.438,E2 -6761.438} C_VEL
LIN {X 0,Y 483.102,Z 401.628,A -85,B 0,C 180,E1 -6761.772,E2 -6761.772} C_VEL
LIN {X 0,Y 483.205,Z 378.212,A -85,B 0,C 180,E1 -6762.151,E2 -6762.151} C_VEL
LIN {X 0,Y 483.235,Z 335.619,A -85,B 0,C 180,E1 -6762.786,E2 -6762.786} C_VEL
LIN {X 0,Y 481.598,Z 324.031,A -85,B 0,C 180,E1 -6763.027,E2 -6763.027} C_VEL
LIN {X 0,Y 481.585,Z 323.283,A -85,B 0,C 180,E1 -6763.116,E2 -6763.116} C_VEL
LIN {X 0,Y 481.93,Z 309.718,A -85,B 0,C 180,E1 -6766.085,E2 -6766.085} C_VEL
LIN {X 0,Y 482.412,Z 296.054,A -85,B 0,C 180,E1 -6769.134,E2 -6769.134} C_VEL
LIN {X 0,Y 482.292,Z 288.846,A -85,B 0,C 180,E1 -6770.778,E2 -6770.778} C_VEL
LIN {X 0,Y 481.718,Z 285.412,A -85,B 0,C 180,E1 -6771.615,E2 -6771.615} C_VEL
LIN {X 0,Y 481.672,Z 285.298,A -85,B 0,C 180,E1 -6775.032,E2 -6775.032} C_VEL
LIN {X 0,Y 481.648,Z 285.301,A -85,B 0,C 180,E1 -6777.834,E2 -6777.834} C_VEL
LIN {X 0,Y 481.638,Z 285.298,A -85,B 0,C 180,E1 -6780.711,E2 -6780.711} C_VEL
LIN {X 0,Y 481.672,Z 285.298,A -85,B 0,C 180,E1 -6783.728,E2 -6783.728} C_VEL
LIN {X 0,Y 481.616,Z 285.302,A -85,B 0,C 180,E1 -6786.747,E2 -6786.747} C_VEL
LIN {X 0,Y 481.653,Z 285.297,A -85,B 0,C 180,E1 -6789.942,E2 -6789.942} C_VEL
LIN {X 0,Y 481.613,Z 285.308,A -85,B 0,C 180,E1 -6793.301,E2 -6793.301} C_VEL
LIN {X 0,Y 481.646,Z 285.299,A -85,B 0,C 180,E1 -6795.641,E2 -6795.641} C_VEL
LIN {X 0,Y 481.616,Z 285.308,A -85,B 0,C 180,E1 -6798.954,E2 -6798.954} C_VEL
LIN {X 0,Y 481.641,Z 285.298,A -85,B 0,C 180,E1 -6801.993,E2 -6801.993} C_VEL
LIN {X 0,Y 481.673,Z 285.296,A -85,B 0,C 180,E1 -6805.316,E2 -6805.316} C_VEL
LIN {X 0,Y 481.63,Z 285.301,A -85,B 0,C 180,E1 -6808.31,E2 -6808.31} C_VEL
LIN {X 0,Y 481.649,Z 285.299,A -85,B 0,C 180,E1 -6811.215,E2 -6811.215} C_VEL
LIN {X 0,Y 481.633,Z 285.3,A -85,B 0,C 180,E1 -6814.039,E2 -6814.039} C_VEL
LIN {X 0,Y 481.642,Z 285.303,A -85,B 0,C 180,E1 -6816.818,E2 -6816.818} C_VEL
LIN {X 0,Y 481.669,Z 285.294,A -85,B 0,C 180,E1 -6819.501,E2 -6819.501} C_VEL
LIN {X 0,Y 481.652,Z 285.3,A -85,B 0,C 180,E1 -6822.156,E2 -6822.156} C_VEL
LIN {X 0,Y 481.718,Z 285.291,A -85,B 0,C 180,E1 -6824.775,E2 -6824.775} C_VEL
LIN {X 0,Y 481.74,Z 285.292,A -85,B 0,C 180,E1 -6828.215,E2 -6828.215} C_VEL
LIN {X 0,Y 481.723,Z 285.289,A -85,B 0,C 180,E1 -6831.611,E2 -6831.611} C_VEL
LIN {X 0,Y 481.765,Z 285.29,A -85,B 0,C 180,E1 -6834.139,E2 -6834.139} C_VEL
LIN {X 0,Y 481.895,Z 285.267,A -85,B 0,C 180,E1 -6837.492,E2 -6837.492} C_VEL
LIN {X 0,Y 481.898,Z 285.274,A -85,B 0,C 180,E1 -6840,E2 -6840} C_VEL
LIN {X 0,Y 481.894,Z 285.268,A -85,B 0,C 180,E1 -6842.508,E2 -6842.508} C_VEL
LIN {X 0,Y 481.763,Z 285.291,A -85,B 0,C 180,E1 -6845.861,E2 -6845.861} C_VEL
LIN {X 0,Y 481.703,Z 285.291,A -85,B 0,C 180,E1 -6848.389,E2 -6848.389} C_VEL
LIN {X 0,Y 481.724,Z 285.295,A -85,B 0,C 180,E1 -6851.786,E2 -6851.786} C_VEL
LIN {X 0,Y 481.717,Z 285.291,A -85,B 0,C 180,E1 -6855.225,E2 -6855.225} C_VEL
LIN {X 0,Y 481.693,Z 285.291,A -85,B 0,C 180,E1 -6858.722,E2 -6858.722} C_VEL
LIN {X 0,Y 481.627,Z 285.306,A -85,B 0,C 180,E1 -6861.396,E2 -6861.396} C_VEL
LIN {X 0,Y 481.634,Z 285.299,A -85,B 0,C 180,E1 -6864.115,E2 -6864.115} C_VEL
LIN {X 0,Y 481.641,Z 285.303,A -85,B 0,C 180,E1 -6867.117,E2 -6867.117} C_VEL
LIN {X 0,Y 481.654,Z 285.298,A -85,B 0,C 180,E1 -6869.743,E2 -6869.743} C_VEL
LIN {X 0,Y 481.642,Z 285.299,A -85,B 0,C 180,E1 -6872.676,E2 -6872.676} C_VEL
LIN {X 0,Y 481.619,Z 285.302,A -85,B 0,C 180,E1 -6875.711,E2 -6875.711} C_VEL
LIN {X 0,Y 481.657,Z 285.301,A -85,B 0,C 180,E1 -6878.86,E2 -6878.86} C_VEL
LIN {X 0,Y 481.607,Z 285.302,A -85,B 0,C 180,E1 -6882.165,E2 -6882.165} C_VEL
LIN {X 0,Y 481.646,Z 285.299,A -85,B 0,C 180,E1 -6884.459,E2 -6884.459} C_VEL
LIN {X 0,Y 481.609,Z 285.31,A -85,B 0,C 180,E1 -6886.856,E2 -6886.856} C_VEL
LIN {X 0,Y 481.649,Z 285.297,A -85,B 0,C 180,E1 -6890.058,E2 -6890.058} C_VEL
LIN {X 0,Y 481.614,Z 285.302,A -85,B 0,C 180,E1 -6893.378,E2 -6893.378} C_VEL
LIN {X 0,Y 481.666,Z 285.299,A -85,B 0,C 180,E1 -6896.327,E2 -6896.327} C_VEL
LIN {X 0,Y 481.638,Z 285.298,A -85,B 0,C 180,E1 -6899.42,E2 -6899.42} C_VEL
LIN {X 0,Y 481.645,Z 285.301,A -85,B 0,C 180,E1 -6902.165,E2 -6902.165} C_VEL
LIN {X 0,Y 481.67,Z 285.298,A -85,B 0,C 180,E1 -6904.968,E2 -6904.968} C_VEL
LIN {X 0,Y 481.74,Z 285.4,A -85,B 0,C 180,E1 -6908.414,E2 -6908.414} C_VEL
LIN {X 0,Y 482.422,Z 289.999,A -85,B 0,C 180,E1 -6909.535,E2 -6909.535} C_VEL
LIN {X 0,Y 482.286,Z 299.758,A -85,B 0,C 180,E1 -6911.742,E2 -6911.742} C_VEL
LIN {X 0,Y 481.762,Z 315.372,A -85,B 0,C 180,E1 -6915.209,E2 -6915.209} C_VEL
LIN {X 0,Y 481.584,Z 323.785,A -85,B 0,C 180,E1 -6917.002,E2 -6917.002} C_VEL
LIN {X 0,Y 482.484,Z 329.877,A -85,B 0,C 180,E1 -6917.153,E2 -6917.153} C_VEL
LIN {X 0,Y 483.441,Z 338.122,A -85,B 0,C 180,E1 -6917.302,E2 -6917.302} C_VEL
LIN {X 0,Y 483.077,Z 399.478,A -85,B 0,C 180,E1 -6918.228,E2 -6918.228} C_VEL
LIN {X 0,Y 482.908,Z 408.429,A -85,B 0,C 180,E1 -6918.457,E2 -6918.457} C_VEL
LIN {X 0,Y 482.79,Z 416.896,A -85,B 0,C 180,E1 -6918.773,E2 -6918.773} C_VEL
LIN {X 0,Y 482.51,Z 425.397,A -85,B 0,C 180,E1 -6919.192,E2 -6919.192} C_VEL
LIN {X 0,Y 482.277,Z 433.728,A -85,B 0,C 180,E1 -6919.717,E2 -6919.717} C_VEL
LIN {X 0,Y 481.99,Z 441.764,A -85,B 0,C 180,E1 -6920.347,E2 -6920.347} C_VEL
LIN {X 0,Y 481.7,Z 450.436,A -85,B 0,C 180,E1 -6921.188,E2 -6921.188} C_VEL
LIN {X 0,Y 481.383,Z 458.94,A -85,B 0,C 180,E1 -6922.239,E2 -6922.239} C_VEL
LIN {X 0,Y 481.239,Z 465.611,A -85,B 0,C 180,E1 -6923.291,E2 -6923.291} C_VEL
LIN {X 0,Y 481.127,Z 469.99,A -85,B 0,C 180,E1 -6924.131,E2 -6924.131} C_VEL
LIN {X 0,Y 480.9,Z 475.15,A -85,B 0,C 180,E1 -6925.39,E2 -6925.39} C_VEL
LIN {X 0,Y 480.917,Z 478.938,A -85,B 0,C 180,E1 -6926.649,E2 -6926.649} C_VEL
LIN {X 0,Y 480.826,Z 480.68,A -85,B 0,C 180,E1 -6927.487,E2 -6927.487} C_VEL
LIN {X 0,Y 480.791,Z 481.928,A -85,B 0,C 180,E1 -6928.325,E2 -6928.325} C_VEL
LIN {X 0,Y 480.757,Z 482.706,A -85,B 0,C 180,E1 -6929.162,E2 -6929.162} C_VEL
LIN {X 0,Y 480.74,Z 483,A -85,B 0,C 180,E1 -6930,E2 -6930} C_VEL
LIN {X 0,Y 480.757,Z 482.705,A -85,B 0,C 180,E1 -6930.838,E2 -6930.838} C_VEL
LIN {X 0,Y 480.791,Z 481.927,A -85,B 0,C 180,E1 -6931.675,E2 -6931.675} C_VEL
LIN {X 0,Y 480.826,Z 480.678,A -85,B 0,C 180,E1 -6932.513,E2 -6932.513} C_VEL
LIN {X 0,Y 480.946,Z 477.786,A -85,B 0,C 180,E1 -6933.77,E2 -6933.77} C_VEL
LIN {X 0,Y 480.9,Z 475.149,A -85,B 0,C 180,E1 -6934.61,E2 -6934.61} C_VEL
LIN {X 0,Y 481.127,Z 469.985,A -85,B 0,C 180,E1 -6935.869,E2 -6935.869} C_VEL
LIN {X 0,Y 481.285,Z 463.181,A -85,B 0,C 180,E1 -6937.13,E2 -6937.13} C_VEL
LIN {X 0,Y 481.487,Z 455.738,A -85,B 0,C 180,E1 -6938.182,E2 -6938.182} C_VEL
LIN {X 0,Y 481.757,Z 448.396,A -85,B 0,C 180,E1 -6939.022,E2 -6939.022} C_VEL
LIN {X 0,Y 482.049,Z 440.531,A -85,B 0,C 180,E1 -6939.758,E2 -6939.758} C_VEL
LIN {X 0,Y 482.346,Z 432.22,A -85,B 0,C 180,E1 -6940.388,E2 -6940.388} C_VEL
LIN {X 0,Y 482.665,Z 421.608,A -85,B 0,C 180,E1 -6941.017,E2 -6941.017} C_VEL
LIN {X 0,Y 482.884,Z 410.072,A -85,B 0,C 180,E1 -6941.491,E2 -6941.491} C_VEL
LIN {X 0,Y 483.061,Z 400.432,A -85,B 0,C 180,E1 -6941.752,E2 -6941.752} C_VEL
LIN {X 0,Y 483.332,Z 336.158,A -85,B 0,C 180,E1 -6942.729,E2 -6942.729} C_VEL
LIN {X 0,Y 481.605,Z 324.059,A -85,B 0,C 180,E1 -6942.976,E2 -6942.976} C_VEL
LIN {X 0,Y 481.571,Z 322.199,A -85,B 0,C 180,E1 -6943.288,E2 -6943.288} C_VEL
LIN {X 0,Y 481.929,Z 309.511,A -85,B 0,C 180,E1 -6946.086,E2 -6946.086} C_VEL
LIN {X 0,Y 482.414,Z 295.848,A -85,B 0,C 180,E1 -6949.134,E2 -6949.134} C_VEL
LIN {X 0,Y 482.273,Z 288.672,A -85,B 0,C 180,E1 -6950.772,E2 -6950.772} C_VEL
LIN {X 0,Y 481.706,Z 285.379,A -85,B 0,C 180,E1 -6951.616,E2 -6951.616} C_VEL
LIN {X 0,Y 481.67,Z 285.298,A -85,B 0,C 180,E1 -6955.032,E2 -6955.032} C_VEL
LIN {X 0,Y 481.646,Z 285.301,A -85,B 0,C 180,E1 -6957.835,E2 -6957.835} C_VEL
LIN {X 0,Y 481.633,Z 285.299,A -85,B 0,C 180,E1 -6960.711,E2 -6960.711} C_VEL
LIN {X 0,Y 481.671,Z 285.298,A -85,B 0,C 180,E1 -6963.728,E2 -6963.728} C_VEL
LIN {X 0,Y 481.613,Z 285.303,A -85,B 0,C 180,E1 -6966.747,E2 -6966.747} C_VEL
LIN {X 0,Y 481.651,Z 285.297,A -85,B 0,C 180,E1 -6969.942,E2 -6969.942} C_VEL
LIN {X 0,Y 481.612,Z 285.308,A -85,B 0,C 180,E1 -6973.302,E2 -6973.302} C_VEL
LIN {X 0,Y 481.645,Z 285.299,A -85,B 0,C 180,E1 -6975.641,E2 -6975.641} C_VEL
LIN {X 0,Y 481.615,Z 285.308,A -85,B 0,C 180,E1 -6978.954,E2 -6978.954} C_VEL
LIN {X 0,Y 481.639,Z 285.298,A -85,B 0,C 180,E1 -6981.993,E2 -6981.993} C_VEL
LIN {X 0,Y 481.671,Z 285.296,A -85,B 0,C 180,E1 -6985.317,E2 -6985.317} C_VEL
LIN {X 0,Y 481.629,Z 285.301,A -85,B 0,C 180,E1 -6988.311,E2 -6988.311} C_VEL
LIN {X 0,Y 481.648,Z 285.299,A -85,B 0,C 180,E1 -6991.215,E2 -6991.215} C_VEL
LIN {X 0,Y 481.632,Z 285.3,A -85,B 0,C 180,E1 -6994.039,E2 -6994.039} C_VEL
LIN {X 0,Y 481.642,Z 285.303,A -85,B 0,C 180,E1 -6996.818,E2 -6996.818} C_VEL
LIN {X 0,Y 481.669,Z 285.294,A -85,B 0,C 180,E1 -6999.502,E2 -6999.502} C_VEL
LIN {X 0,Y 481.652,Z 285.3,A -85,B 0,C 180,E1 -7002.156,E2 -7002.156} C_VEL
LIN {X 0,Y 481.717,Z 285.291,A -85,B 0,C 180,E1 -7004.775,E2 -7004.775} C_VEL
LIN {X 0,Y 481.739,Z 285.292,A -85,B 0,C 180,E1 -7008.215,E2 -7008.215} C_VEL
LIN {X 0,Y 481.708,Z 285.29,A -85,B 0,C 180,E1 -7011.611,E2 -7011.611} C_VEL
LIN {X 0,Y 481.764,Z 285.29,A -85,B 0,C 180,E1 -7014.139,E2 -7014.139} C_VEL
LIN {X 0,Y 481.895,Z 285.267,A -85,B 0,C 180,E1 -7017.492,E2 -7017.492} C_VEL
LIN {X 0,Y 481.898,Z 285.274,A -85,B 0,C 180,E1 -7020,E2 -7020} C_VEL
LIN {X 0,Y 481.895,Z 285.268,A -85,B 0,C 180,E1 -7022.508,E2 -7022.508} C_VEL
LIN {X 0,Y 481.764,Z 285.291,A -85,B 0,C 180,E1 -7025.861,E2 -7025.861} C_VEL
LIN {X 0,Y 481.7,Z 285.292,A -85,B 0,C 180,E1 -7028.389,E2 -7028.389} C_VEL
LIN {X 0,Y 481.724,Z 285.295,A -85,B 0,C 180,E1 -7031.786,E2 -7031.786} C_VEL
LIN {X 0,Y 481.717,Z 285.291,A -85,B 0,C 180,E1 -7035.225,E2 -7035.225} C_VEL
LIN {X 0,Y 481.693,Z 285.291,A -85,B 0,C 180,E1 -7038.723,E2 -7038.723} C_VEL
LIN {X 0,Y 481.627,Z 285.306,A -85,B 0,C 180,E1 -7041.396,E2 -7041.396} C_VEL
LIN {X 0,Y 481.635,Z 285.299,A -85,B 0,C 180,E1 -7044.115,E2 -7044.115} C_VEL
LIN {X 0,Y 481.641,Z 285.302,A -85,B 0,C 180,E1 -7047.117,E2 -7047.117} C_VEL
LIN {X 0,Y 481.641,Z 285.3,A -85,B 0,C 180,E1 -7049.744,E2 -7049.744} C_VEL
LIN {X 0,Y 481.641,Z 285.299,A -85,B 0,C 180,E1 -7052.677,E2 -7052.677} C_VEL
LIN {X 0,Y 481.62,Z 285.302,A -85,B 0,C 180,E1 -7055.711,E2 -7055.711} C_VEL
LIN {X 0,Y 481.626,Z 285.305,A -85,B 0,C 180,E1 -7058.864,E2 -7058.864} C_VEL
LIN {X 0,Y 481.614,Z 285.301,A -85,B 0,C 180,E1 -7061.909,E2 -7061.909} C_VEL
LIN {X 0,Y 481.648,Z 285.299,A -85,B 0,C 180,E1 -7064.459,E2 -7064.459} C_VEL
LIN {X 0,Y 481.61,Z 285.31,A -85,B 0,C 180,E1 -7066.856,E2 -7066.856} C_VEL
LIN {X 0,Y 481.651,Z 285.297,A -85,B 0,C 180,E1 -7070.058,E2 -7070.058} C_VEL
LIN {X 0,Y 481.615,Z 285.302,A -85,B 0,C 180,E1 -7073.378,E2 -7073.378} C_VEL
LIN {X 0,Y 481.667,Z 285.298,A -85,B 0,C 180,E1 -7076.328,E2 -7076.328} C_VEL
LIN {X 0,Y 481.615,Z 285.301,A -85,B 0,C 180,E1 -7079.425,E2 -7079.425} C_VEL
LIN {X 0,Y 481.643,Z 285.301,A -85,B 0,C 180,E1 -7082.165,E2 -7082.165} C_VEL
LIN {X 0,Y 481.671,Z 285.298,A -85,B 0,C 180,E1 -7084.968,E2 -7084.968} C_VEL
LIN {X 0,Y 481.651,Z 285.279,A -85,B 0,C 180,E1 -7087.94,E2 -7087.94} C_VEL
LIN {X 0,Y 481.391,Z 285.827,A -85,B 0,C 180,E1 -7088.403,E2 -7088.403} C_VEL
LIN {X 0,Y 480.697,Z 287.186,A -85,B 0,C 180,E1 -7088.84,E2 -7088.84} C_VEL
LIN {X 0,Y 475.665,Z 296.906,A -85,B 0,C 180,E1 -7090.869,E2 -7090.869} C_VEL
LIN {X 0,Y 475.335,Z 298.788,A -85,B 0,C 180,E1 -7091.29,E2 -7091.29} C_VEL
LIN {X 0,Y 474.813,Z 313.215,A -85,B 0,C 180,E1 -7094.549,E2 -7094.549} C_VEL
LIN {X 0,Y 474.55,Z 323.723,A -85,B 0,C 180,E1 -7096.844,E2 -7096.844} C_VEL
LIN {X 0,Y 475.218,Z 328.173,A -85,B 0,C 180,E1 -7096.974,E2 -7096.974} C_VEL
LIN {X 0,Y 476.466,Z 338.038,A -85,B 0,C 180,E1 -7097.158,E2 -7097.158} C_VEL
LIN {X 0,Y 476.207,Z 399.558,A -85,B 0,C 180,E1 -7098.103,E2 -7098.103} C_VEL
LIN {X 0,Y 475.982,Z 408.679,A -85,B 0,C 180,E1 -7098.341,E2 -7098.341} C_VEL
LIN {X 0,Y 475.777,Z 418.288,A -85,B 0,C 180,E1 -7098.713,E2 -7098.713} C_VEL
LIN {X 0,Y 475.487,Z 428.346,A -85,B 0,C 180,E1 -7099.246,E2 -7099.246} C_VEL
LIN {X 0,Y 475.143,Z 438.784,A -85,B 0,C 180,E1 -7099.992,E2 -7099.992} C_VEL
LIN {X 0,Y 474.799,Z 446.945,A -85,B 0,C 180,E1 -7100.737,E2 -7100.737} C_VEL
LIN {X 0,Y 474.539,Z 453.678,A -85,B 0,C 180,E1 -7101.483,E2 -7101.483} C_VEL
